// TwinCAT 3 PLC project PLC1
// ProgramVersion: 3.1.4026.16
// CompilerDefines: VISU_USEPROPERTYINFO
// libraries:
//   SH_Light, * (StroemHansen)
//   Tc2_EnOcean, * (Beckhoff Automation GmbH)
//   Tc2_Standard, * (Beckhoff Automation GmbH)
//   Tc2_System, * (Beckhoff Automation GmbH)
//   Tc2_Utilities, * (Beckhoff Automation GmbH)
//   Tc3_DALI, * (Beckhoff Automation GmbH)
//   Tc3_System_DK, * (Beckhoff - DK)
//   VisuDialogs, * (System)
// project tree:
//   DUTs/DALI/ E_DALIExtendedFadeTime.TcTLEO (not stored), ST_DALI102Parameters.TcDUT (not stored), ST_DALI103Parameters.TcDUT, ST_DALIMemoryBank.TcDUT (not stored), ST_DALI_GrpAssignment.TcDUT (not stored), ST_GroupSort.TcDUT (not stored)
//   DUTs/EnOcean/ ST_ReadSAB05.TcDUT (not stored), ST_WriteSAB05.TcDUT (not stored)
//   / FastTask.TcTTO (not stored), GlobalTextList.TcGTLO, PlcTask.TcTTO (not stored), Visualization Manager.TcVMO (not stored)
//   GVLs/ GVL_AHDataModbus.TcGVL (not stored), GVL_EnOcean.TcGVL, GVL_Skalering.TcGVL
//   POUs/01_System/01_System/GVLs/ GVL_EtherCAT.TcGVL (not stored)
//   POUs/01_System/01_System/ P_SystemDK.TcPOU (not stored)
//   POUs/AHModbusComm/ P_AHModbusComm.TcPOU
//   POUs/Alle_Rum/Gange/P_Gang_1_108/ P_Gang_1_108.TcPOU, Visualization_1_108.TcVIS (excluded from build)
//   POUs/Alle_Rum/Gange/P_Gang_1_111A/ P_Gang_1_111A.TcPOU, Visualization_1_111A.TcVIS (excluded from build)
//   POUs/Alle_Rum/Rum_Med_DALI_Pir/ P_Lys_Grp0.TcPOU (not stored) (excluded from build)
//   POUs/Alle_Rum/Rum_Med_DALI_Pir/Rum_1_111D/ P_Rum_1_111D.TcPOU, Visualization_1_111D.TcVIS (excluded from build)
//   POUs/Alle_Rum/Rum_Med_DALI_Pir/Rum_1_111E/ P_Rum_1_111E.TcPOU, Visualization_1.TcVIS (excluded from build)
//   POUs/Alle_Rum/Rum_Med_DALI_Pir/Rum_1_111C/ P_Rum_1_111C.TcPOU, Visualization_1_111C.TcVIS (excluded from build)
//   POUs/Alle_Rum/Rum_Med_DALI_Pir/Rum_1_115/ P_Rum_1_115.TcPOU, Visualization_1_115.TcVIS (excluded from build)
//   POUs/Alle_Rum/Rum_Med_DALI_Pir/Rum_1_118/ P_Rum_1_118.TcPOU, Visualization_1_118.TcVIS (excluded from build)
//   POUs/Alle_Rum/Rum_Med_DALI_Pir/Rum_1_106/ P_Rum_1_106.TcPOU, Visualization_1_106.TcVIS (excluded from build)
//   POUs/Alle_Rum/Trapper/ P_Trappe_T1.TcPOU
//   POUs/DALI/DALI_Setup/ DALI_Commissioning.TcPOU (not stored)
//   POUs/DALI/DALI_Setup/FBs/ FB_Part102Addressing.TcPOU (not stored), FB_Part102Commands.TcPOU (not stored), FB_Part102Groups.TcPOU (not stored), FB_Part102MemoryPages.TcPOU, FB_Part102Parameters.TcPOU, FB_Part102Scenes.TcPOU (not stored), FB_Part102SetFading.TcPOU, FB_Part103Addressing.TcPOU (not stored), FB_Part103MemoryPages.TcPOU (not stored), FB_Part103Identify.TcPOU (not stored), FB_Part103Parameters.TcPOU (not stored), FB_Part202Emergency.TcPOU (not stored), FB_Part205Incandescent.TcPOU (not stored), FB_Part207LED.TcPOU (not stored), FB_Part208Switching.TcPOU (not stored), FB_Part300GenericDevice.TcPOU (not stored), FB_Part301PushButton.TcPOU (not stored), FB_Part302AbsoluteInputDevice.TcPOU (not stored), FB_Part303OccupancySensor.TcPOU (not stored), FB_Part304LightSensor.TcPOU (not stored), GearType.TcPOU (not stored)
//   POUs/DALI/DALI_Setup/GVLs/ GVL_Internal.TcGVL (not stored)
//   POUs/DALI/DALI_Setup/VISUs/TextLists/ CommandOnTerminalEvent.TcTLO (not stored), DimmingCurve.TcTLO, EventPriority.TcTLO (not stored), EventScheme.TcTLO (not stored), ExtendedFadeTime.TcTLO (not stored), FadeRate.TcTLO (not stored), FadeTime.TcTLO (not stored), FastFadeTime.TcTLO (not stored), TextList_Dialogs.TcTLO (not stored)
//   POUs/DALI/DALI_Setup/VISUs/ Visu_DALICommissioning.TcVIS (not stored)
//   POUs/DALI/DALI_Setup/VISUs/Visu_DALICommissioning/ Visu_KL6821Configuration.TcVIS (not stored) (excluded from build), Visu_Part102Addressing.TcVIS (not stored), Visu_Part102Commands.TcVIS (not stored), Visu_Part102Groups.TcVIS (not stored), Visu_Part102MemoryBank.TcVIS, Visu_Part102Parameters.TcVIS, Visu_Part102Scenes.TcVIS (not stored), Visu_Part102SetFading.TcVIS (not stored), Visu_Part103Addressing.TcVIS (not stored), Visu_Part103MemoryBank.TcVIS, Visu_Part103Identify.TcVIS (not stored), Visu_Part103Parameters.TcVIS (not stored), Visu_Part202.TcVIS (not stored), Visu_Part202Commands.TcVIS, Visu_Part202Parameters.TcVIS (not stored), Visu_Part202Status.TcVIS (not stored), Visu_Part205.TcVIS (not stored), Visu_Part205Parameters.TcVIS (not stored), Visu_Part205Status.TcVIS, Visu_Part207.TcVIS (not stored), Visu_Part207Parameters.TcVIS (not stored), Visu_Part207Status.TcVIS, Visu_Part208Switching.TcVIS (not stored), Visu_Part300GenericDevice.TcVIS (not stored), Visu_Part301PushButton.TcVIS (not stored), Visu_Part302AbsoluteInputDevice.TcVIS, Visu_Part303OccupancySensor.TcVIS, Visu_Part304LightSensor.TcVIS, Visu_Welcome.TcVIS (not stored)
//   POUs/DALI/PRGs/Background/ P_DALI_Background.TcPOU (not stored)
//   POUs/DALI/PRGs/Diag/ P_DALI_DIAG.TcPOU (not stored)
//   POUs/DALI/PRGs/EnergyData/ P_DALI_Energy_Firmware_Test.TcPOU (not stored) (excluded from build), P_DALI_Energy_Line.TcPOU (not stored)
//   POUs/EnOcean/ P_EnOcean.TcPOU
//   POUs/ MAIN.TcPOU
//   POUs/Tester/ P_DALI2_Test.TcPOU (not stored) (excluded from build), P_Test_TypeA.TcPOU (not stored) (excluded from build), Visualization.TcVIS (excluded from build)
// real-time tasks:
//   TASK PlcTask: cycle T#40ms, priority 21, ADS port 350
//   TASK FastTask: cycle T#4ms, priority 20, ADS port 351
// I/O:
//   DEVICE Device 1 (Beckhoff CCAT)
//   DEVICE Device 3 (CX-BK)
//     Box 1 (CX-BK)
// variable links:
//   PLC1/PLC1 Instance <-> Device 3 (CX-BK)/Box 1 (CX-BK)
//     FastTask Inputs/P_DALI_Background.arrKL6821InData[1] @bit 16 <-> Term 5 (KL6821)/Channel 1/Data In 0
//     FastTask Inputs/P_DALI_Background.arrKL6821InData[1] @bit 24 <-> Term 5 (KL6821)/Channel 1/Data In 1
//     FastTask Inputs/P_DALI_Background.arrKL6821InData[1] @bit 32 <-> Term 5 (KL6821)/Channel 1/Data In 2
//     FastTask Inputs/P_DALI_Background.arrKL6821InData[1] @bit 40 <-> Term 5 (KL6821)/Channel 1/Data In 3
//     FastTask Inputs/P_DALI_Background.arrKL6821InData[2] @bit 16 <-> Term 6 (KL6821)/Channel 1/Data In 0
//     FastTask Inputs/P_DALI_Background.arrKL6821InData[2] @bit 24 <-> Term 6 (KL6821)/Channel 1/Data In 1
//     FastTask Inputs/P_DALI_Background.arrKL6821InData[2] @bit 32 <-> Term 6 (KL6821)/Channel 1/Data In 2
//     FastTask Inputs/P_DALI_Background.arrKL6821InData[2] @bit 40 <-> Term 6 (KL6821)/Channel 1/Data In 3
//     FastTask Inputs/P_DALI_Background.arrKL6821InData[1] <-> Term 5 (KL6821)/Channel 1/State
//     FastTask Inputs/P_DALI_Background.arrKL6821InData[2] <-> Term 6 (KL6821)/Channel 1/State
//     FastTask Inputs/P_EnOcean.stKL6581_in @bit 8 <-> Term 3 (KL6581)/Channel 1/Input CNODE
//     FastTask Inputs/P_EnOcean.stKL6581_in @bit {24..48 step 8} <-> Term 3 (KL6581)/Channel 1/Input DB{0..3}  (4 links)
//     FastTask Inputs/P_EnOcean.stKL6581_in @bit {56..80 step 8} <-> Term 3 (KL6581)/Channel 1/Input ID{0..3}  (4 links)
//     FastTask Inputs/P_EnOcean.stKL6581_in @bit 16 <-> Term 3 (KL6581)/Channel 1/Input ORG
//     FastTask Inputs/P_EnOcean.stKL6581_in @bit 88 <-> Term 3 (KL6581)/Channel 1/Input STATUS
//     FastTask Inputs/P_EnOcean.stKL6581_in <-> Term 3 (KL6581)/Channel 1/Status
//     FastTask Outputs/P_DALI_Background.arrKL6821OutData[1] <-> Term 5 (KL6821)/Channel 1/Ctrl
//     FastTask Outputs/P_DALI_Background.arrKL6821OutData[2] <-> Term 6 (KL6821)/Channel 1/Ctrl
//     FastTask Outputs/P_DALI_Background.arrKL6821OutData[1] @bit 16 <-> Term 5 (KL6821)/Channel 1/Data Out 0
//     FastTask Outputs/P_DALI_Background.arrKL6821OutData[1] @bit 24 <-> Term 5 (KL6821)/Channel 1/Data Out 1
//     FastTask Outputs/P_DALI_Background.arrKL6821OutData[1] @bit 32 <-> Term 5 (KL6821)/Channel 1/Data Out 2
//     FastTask Outputs/P_DALI_Background.arrKL6821OutData[1] @bit 40 <-> Term 5 (KL6821)/Channel 1/Data Out 3
//     FastTask Outputs/P_DALI_Background.arrKL6821OutData[2] @bit 16 <-> Term 6 (KL6821)/Channel 1/Data Out 0
//     FastTask Outputs/P_DALI_Background.arrKL6821OutData[2] @bit 24 <-> Term 6 (KL6821)/Channel 1/Data Out 1
//     FastTask Outputs/P_DALI_Background.arrKL6821OutData[2] @bit 32 <-> Term 6 (KL6821)/Channel 1/Data Out 2
//     FastTask Outputs/P_DALI_Background.arrKL6821OutData[2] @bit 40 <-> Term 6 (KL6821)/Channel 1/Data Out 3
//     FastTask Outputs/P_EnOcean.stKL6581_out <-> Term 3 (KL6581)/Channel 1/Control
//     FastTask Outputs/P_EnOcean.stKL6581_out @bit 8 <-> Term 3 (KL6581)/Channel 1/Output CNODE
//     FastTask Outputs/P_EnOcean.stKL6581_out @bit {24..48 step 8} <-> Term 3 (KL6581)/Channel 1/Output DB{0..3}  (4 links)
//     FastTask Outputs/P_EnOcean.stKL6581_out @bit {56..80 step 8} <-> Term 3 (KL6581)/Channel 1/Output ID{0..3}  (4 links)
//     FastTask Outputs/P_EnOcean.stKL6581_out @bit 16 <-> Term 3 (KL6581)/Channel 1/Output ORG
//     FastTask Outputs/P_EnOcean.stKL6581_out @bit 88 <-> Term 3 (KL6581)/Channel 1/Output STATUS
//     PlcTask Inputs/MAIN.nCX8200_State <-> Inputs/State
//     PlcTask Inputs/P_Trappe_T1.bDigitalPir <-> Term 4 (KL1408)/Channel 1/Input
//     PlcTask Outputs/P_Trappe_T1.bTrappelysNC <-> Term 2 (KL2012)/Channel 1/Output

// ---- DUTs/DALI/ST_DALI103Parameters.TcDUT
TYPE ST_DALI103Parameters :
STRUCT	
	//nShortAddress			:	BYTE;
	nOperatingMode			:	BYTE;
	sInstanceType0			:	STRING;	
	sInstanceType1			:	STRING;
	sInstanceType2			:	STRING;
	sInstanceType3			:	STRING;
	sInstanceType4			:	STRING;
END_STRUCT
END_TYPE

// ---- GVLs/GVL_EnOcean.TcGVL
{attribute 'qualified_only'}
VAR_GLOBAL
	strEnOceanSwitch_Gang_1_108: Tc2_EnOcean.STR_EnOceanSwitch;
	strEnOceanSwitch_Rum_1_106: Tc2_EnOcean.STR_EnOceanSwitch;
	strEnOceanSwitch_Rum_1_111E: Tc2_EnOcean.STR_EnOceanSwitch;
	strEnOceanSwitch_Rum_1_115_Gang: Tc2_EnOcean.STR_EnOceanSwitch;
	strEnOceanSwitch_Rum_1_115_Ydermur: Tc2_EnOcean.STR_EnOceanSwitch;
	strEnOceanSwitch_Rum_1_118: Tc2_EnOcean.STR_EnOceanSwitch;
	//strEnOceanSwitch_Rum_1_118: Tc2_EnOcean.STR_EnOceanSwitch;
END_VAR

// ---- GVLs/GVL_Skalering.TcGVL
//{attribute 'qualified_only'}
VAR_GLOBAL
fMeassure_Zone1 :REAL:= 604; 
fRead_Zone1     :REAL:= 340;

fMeassure_Zone2 :REAL:=611;
fRead_Zone2     :REAL:=374;

fMeassure_Zone3 :REAL:=986;
fRead_Zone3     :REAL:=524;

fMeassure_Zone4 :REAL:=770;
fRead_Zone4     :REAL:=506;

fMeassure_Zone5 :REAL:=734;
fRead_Zone5     :REAL:=395;

fMeassure_Zone6 :REAL:=890;
fRead_Zone6     :REAL:=476;

fMeassure_Zone7 :REAL:=710;
fRead_Zone7     :REAL:=654;

fMeassure_Zone8 :REAL:=604;
fRead_Zone8     :REAL:=292;

fMeassure_Zone9 :REAL:=572;
fRead_Zone9     :REAL:=348;

fMeassure_Zone10:REAL:= 790;
fRead_Zone10    :REAL:=434;

fMeassure_Zone11 :REAL:=691;
fRead_Zone11     :REAL:=426;

END_VAR

// ---- POUs/AHModbusComm/P_AHModbusComm.TcPOU
PROGRAM P_AHModbusComm
VAR
	arrfbReadAHPirData	: ARRAY[1..GVL_AHDataModbus.byNumberOfAH_Neighbors] OF SH_Light.FB_ReadAHPirData;
	arrReadAHPirData		: ARRAY[1..GVL_AHDataModbus.byNumberOfAH_Neighbors] OF BOOL;
	
	arrfbTriggerPulses			: ARRAY[1..GVL_AHDataModbus.byNumberOfAH_Neighbors] OF SH_Light.FB_ClockPulse;
	arrGeneratePulses			: ARRAY[1..GVL_AHDataModbus.byNumberOfAH_Neighbors] OF BOOL := [GVL_AHDataModbus.byNumberOfAH_Neighbors(TRUE)];
	tTimeInterval					: TIME := T#1S;
	tPulseTime					: TIME := T#1S;
	
	byLineId						: BYTE;
	byAHId						: BYTE;
		fbWritePirDelayTime		: R_TRIG;
	bRunOverrideOnce		: BOOL := FALSE;
	bEnableDelayTimeOverride : BOOL := FALSE;
	uiPirOffDelayTimeAllRooms : UINT := 30;
	
END_VAR

VAR CONSTANT
	arrnMBAddr					: ARRAY[1..GVL_AHDataModbus.byNumberOfAH_Neighbors] OF WORD := [GVL_AHDataModbus.byNumberOfAH_Neighbors(12588)]; //modbus-adresser (%MB600=>12588 default)
	arrstNeighborIPAddr		: ARRAY[1..GVL_AHDataModbus.byNumberOfAH_Neighbors] OF SH_Light.ST_NeighborIP := [
																						(sPLCName := 'AH1-1', sIP := '172.24.195.161', IsNeighbor := FALSE), 
																				     	(sPLCName := 'AH1-2', sIP := '172.24.195.162', IsNeighbor := FALSE), 
																						(sPLCName := 'AH1-3', sIP := '172.24.195.163', IsNeighbor := FALSE),
																						(sPLCName := 'AH2-1', sIP := '172.24.195.164', IsNeighbor := FALSE),
																					    (sPLCName := 'AH2-2', sIP := '172.24.195.165', IsNeighbor := FALSE),
																						(sPLCName := 'AH2-3', sIP := '172.24.195.166', IsNeighbor := FALSE),
																				        (sPLCName := 'AH2-4', sIP := '172.24.195.167', IsNeighbor := FALSE),
																						(sPLCName := 'AH2-5', sIP := '172.24.195.168', IsNeighbor := FALSE),
																						(sPLCName := 'AH3-2', sIP := '172.24.195.169', IsNeighbor := FALSE),
																						(sPLCName := 'AH3-3', sIP := '172.24.195.170', IsNeighbor := FALSE),
																			         	(sPLCName := 'AH3-4', sIP := '172.24.195.171', IsNeighbor := FALSE),
																						(sPLCName := 'AH3-5', sIP := '172.24.195.172', IsNeighbor := FALSE),
																						(sPLCName := 'AH4-1', sIP := '172.24.195.173', IsNeighbor := FALSE),
																						(sPLCName := 'AH4-2', sIP := '172.24.195.174', IsNeighbor := FALSE),
																						(sPLCName := 'AH4-3', sIP := '172.24.195.175', IsNeighbor := FALSE),
																			            (sPLCName := 'AH4-4', sIP := '172.24.195.176', IsNeighbor := FALSE),
																						(sPLCName := 'AH4-5', sIP := '172.24.195.177', IsNeighbor := FALSE),
																						(sPLCName := 'AH5-1', sIP := '172.24.195.178', IsNeighbor := FALSE),
																					    (sPLCName := 'AH5-2', sIP := '172.24.195.179', IsNeighbor := FALSE), 
																						(sPLCName := 'AH5-3', sIP := '172.24.195.180', IsNeighbor := FALSE),
																						(sPLCName := 'AH5-4', sIP := '172.24.195.181', IsNeighbor := FALSE),
																						(sPLCName := 'AH5-5', sIP := '172.24.195.182', IsNeighbor := FALSE),
																						(sPLCName := 'AH6-1', sIP := '172.24.195.183', IsNeighbor := FALSE),
																				        (sPLCName := 'AH6-2', sIP := '172.24.195.184', IsNeighbor := FALSE),//Local must be false
																				(sPLCName := 'AH6-3', sIP := '172.24.195.185', IsNeighbor := FALSE)];
																					//	(sPLCName := 'AH3-1', sIP := '172.24.195.186', IsNeighbor := TRUE) //when ready
END_VAR

A_AHNeighborRoomsPirIn();
A_AHNeighborRoomsPirOut();
A_DALILineShrtAddrErr();
A_DelayTimeAllRooms();

ACTION A_AHNeighborRoomsPirIn:
FOR byAHId := 1 TO GVL_AHDataModbus.byNumberOfAH_Neighbors DO
	IF arrstNeighborIPAddr[byAHId].IsNeighbor THEN
		//Generate Pulses
		arrfbTriggerPulses[byAHId](bGenerateClockPulses:= arrGeneratePulses[byAHId], tTimeInterval:= tTimeInterval, tPulseTime:= tPulseTime);
		arrReadAHPirData[byAHId]:= arrfbTriggerPulses[byAHId].bPulse;
		//Read data
		arrfbReadAHPirData[byAHId](	bReadAHPirData				:=	arrReadAHPirData[byAHId],
														sIPAddr							:=	arrstNeighborIPAddr[byAHId].sIP,
														nMBAddr							:=	arrnMBAddr[byAHId],
														nMBDataBuffer				:=	GVL_AHDataModbus.arrAH_NeighborRoomsPir_In[byAHId],
														arrAH_NeighborRoomsPir	=>GVL_AHDataModbus.arrAH_NeighborRoomsPir[byAHId]);
	END_IF
END_FOR
END_ACTION

ACTION A_AHNeighborRoomsPirOut:
//GVL_AHDataModbus.nAH_NeighborRoomsPir_Out.0 := P_Gang_4_413.bPirActive_MB;
//GVL_AHDataModbus.nAH_NeighborRoomsPir_Out.1 := P_Gang_7_401.bPirActive_MB;
//GVL_AHDataModbus.nAH_NeighborRoomsPir_Out.2 := P_Gang_5_441.bPirActive_MB;
//GVL_AHDataModbus.nAH_NeighborRoomsPir_Out.3 := P_Rum_4_424.bPirActive_MB;
//GVL_AHDataModbus.nAH_NeighborRoomsPir_Out.4 := P_Rum_4_426.bPirActive_MB;
//GVL_AHDataModbus.nAH_NeighborRoomsPir_Out.5 := 
//GVL_AHDataModbus.nAH_NeighborRoomsPir_Out.6 :=
//GVL_AHDataModbus.nAH_NeighborRoomsPir_Out.7 := 
//GVL_AHDataModbus.nAH_NeighborRoomsPir_Out.8 :=
//GVL_AHDataModbus.nAH_NeighborRoomsPir_Out.9 := 
//GVL_AHDataModbus.nAH_NeighborRoomsPir_Out.10 :=
//GVL_AHDataModbus.nAH_NeighborRoomsPir_Out.11 := 
//GVL_AHDataModbus.nAH_NeighborRoomsPir_Out.12 := 
//GVL_AHDataModbus.nAH_NeighborRoomsPir_Out.13 := 
//GVL_AHDataModbus.nAH_NeighborRoomsPir_Out.14 := 
//GVL_AHDataModbus.nAH_NeighborRoomsPir_Out.15 :=
END_ACTION

ACTION A_DALILineShrtAddrErr:
FOR  byLineId := 1 TO SH_Light.DALI_Param.MAX_DALIV2_LINES DO
	GVL_AHDataModbus.arrDALILineShrtAddrErr[byLineId] :=  TO_UINT(SH_Light.GVL_DALI_LatestError.arrLineShrtAddr[byLineId]);
END_FOR
END_ACTION

ACTION A_DelayTimeAllRooms:

fbWritePirDelayTime(CLK := GVL_AHDataModbus.uiPirOffDelayTimeAllRooms_MB<>uiPirOffDelayTimeAllRooms);

IF fbWritePirDelayTime.Q THEN
	bRunOverrideOnce := TRUE;
	bEnableDelayTimeOverride := TRUE;
	
//Indsæt kode
P_Gang_1_108.fbWritePirDelayTIme(bEnableOverride := bEnableDelayTimeOverride, nOverRideValue := GVL_AHDataModbus.uiPirOffDelayTimeAllRooms_MB, nValIn1 := GVL_AHDataModbus.uiPirOffDelayTimeAllRooms_MB, nValIn2 := uiPirOffDelayTimeAllRooms);
P_RUM_1_106.fbWritePirDelayTIme(bEnableOverride := bEnableDelayTimeOverride, nOverRideValue := GVL_AHDataModbus.uiPirOffDelayTimeAllRooms_MB, nValIn1 := GVL_AHDataModbus.uiPirOffDelayTimeAllRooms_MB, nValIn2 := uiPirOffDelayTimeAllRooms);
P_Rum_1_111E.fbWritePirDelayTIme(bEnableOverride := bEnableDelayTimeOverride, nOverRideValue := GVL_AHDataModbus.uiPirOffDelayTimeAllRooms_MB, nValIn1 := GVL_AHDataModbus.uiPirOffDelayTimeAllRooms_MB, nValIn2 := uiPirOffDelayTimeAllRooms);
P_Rum_1_115.fbWritePirDelayTIme(bEnableOverride := bEnableDelayTimeOverride, nOverRideValue := GVL_AHDataModbus.uiPirOffDelayTimeAllRooms_MB, nValIn1 := GVL_AHDataModbus.uiPirOffDelayTimeAllRooms_MB, nValIn2 := uiPirOffDelayTimeAllRooms);
P_Rum_1_118.fbWritePirDelayTIme(bEnableOverride := bEnableDelayTimeOverride, nOverRideValue := GVL_AHDataModbus.uiPirOffDelayTimeAllRooms_MB, nValIn1 := GVL_AHDataModbus.uiPirOffDelayTimeAllRooms_MB, nValIn2 := uiPirOffDelayTimeAllRooms);
P_Rum_1_111D.fbWritePirDelayTIme(bEnableOverride := bEnableDelayTimeOverride, nOverRideValue := GVL_AHDataModbus.uiPirOffDelayTimeAllRooms_MB, nValIn1 := GVL_AHDataModbus.uiPirOffDelayTimeAllRooms_MB, nValIn2 := uiPirOffDelayTimeAllRooms);
P_Gang_1_111A.fbWritePirDelayTIme(bEnableOverride := bEnableDelayTimeOverride, nOverRideValue := GVL_AHDataModbus.uiPirOffDelayTimeAllRooms_MB, nValIn1 := GVL_AHDataModbus.uiPirOffDelayTimeAllRooms_MB, nValIn2 := uiPirOffDelayTimeAllRooms);




ELSE
	IF bRunOverrideOnce THEN
		bEnableDelayTimeOverride := FALSE;
		
		//Indsæt kode
P_Gang_1_108.fbWritePirDelayTIme(bEnableOverride := bEnableDelayTimeOverride, nOverRideValue := GVL_AHDataModbus.uiPirOffDelayTimeAllRooms_MB, nValIn1 := GVL_AHDataModbus.uiPirOffDelayTimeAllRooms_MB, nValIn2 := uiPirOffDelayTimeAllRooms);
P_RUM_1_106.fbWritePirDelayTIme(bEnableOverride := bEnableDelayTimeOverride, nOverRideValue := GVL_AHDataModbus.uiPirOffDelayTimeAllRooms_MB, nValIn1 := GVL_AHDataModbus.uiPirOffDelayTimeAllRooms_MB, nValIn2 := uiPirOffDelayTimeAllRooms);
P_Rum_1_111E.fbWritePirDelayTIme(bEnableOverride := bEnableDelayTimeOverride, nOverRideValue := GVL_AHDataModbus.uiPirOffDelayTimeAllRooms_MB, nValIn1 := GVL_AHDataModbus.uiPirOffDelayTimeAllRooms_MB, nValIn2 := uiPirOffDelayTimeAllRooms);
P_Rum_1_115.fbWritePirDelayTIme(bEnableOverride := bEnableDelayTimeOverride, nOverRideValue := GVL_AHDataModbus.uiPirOffDelayTimeAllRooms_MB, nValIn1 := GVL_AHDataModbus.uiPirOffDelayTimeAllRooms_MB, nValIn2 := uiPirOffDelayTimeAllRooms);
P_Rum_1_118.fbWritePirDelayTIme(bEnableOverride := bEnableDelayTimeOverride, nOverRideValue := GVL_AHDataModbus.uiPirOffDelayTimeAllRooms_MB, nValIn1 := GVL_AHDataModbus.uiPirOffDelayTimeAllRooms_MB, nValIn2 := uiPirOffDelayTimeAllRooms);
P_Rum_1_111D.fbWritePirDelayTIme(bEnableOverride := bEnableDelayTimeOverride, nOverRideValue := GVL_AHDataModbus.uiPirOffDelayTimeAllRooms_MB, nValIn1 := GVL_AHDataModbus.uiPirOffDelayTimeAllRooms_MB, nValIn2 := uiPirOffDelayTimeAllRooms);
P_Gang_1_111A.fbWritePirDelayTIme(bEnableOverride := bEnableDelayTimeOverride, nOverRideValue := GVL_AHDataModbus.uiPirOffDelayTimeAllRooms_MB, nValIn1 := GVL_AHDataModbus.uiPirOffDelayTimeAllRooms_MB, nValIn2 := uiPirOffDelayTimeAllRooms);

		bRunOverrideOnce := FALSE;
		
		
	END_IF
END_IF
END_ACTION

END_PROGRAM

// ---- POUs/Alle_Rum/Gange/P_Gang_1_108/P_Gang_1_108.TcPOU
PROGRAM P_Gang_1_108
VAR
//Light

	fbLys		: FB_Light_Type_B;
	
	stDaliSetup	: SH_Light.ST_DALI_RoomSetup := (		byShrtAdr_Prim := 25, 
														byGrpAdr_Prim := 4, 
														eMod_Prim := E_DALIAddressType.Group, 
														//byShrtAdr_Sec := 1, 
														//byGrpAdr_Sec := 1, 
														//eMod_Sec := E_DALIAddressType.Short, 
														//byShrtAdr_Supl := 1, 
														DALI_LINE_NUM_PRIM := 1, 
														DALI_LINE_NUM_SEC := 0, 
														DALI_LINE_NUM_SUPL := 0);
	stLiveData				: SH_Light.ST_LiveData;
	bRunTuning					: BOOL;
	
	bTopButtonZone1				: BOOL;
	bTopButtonZone1_Visu		: BOOL;
	bBottomButtonZone1			: BOOL;
	bBottomButtonZone1_Visu	    : BOOL;
	bButtonZone2				: BOOL;
	bNeighborRoomsPir		    : BOOL;
	fLuxOn				     	: REAL;
	fLuxDim						: REAL;
	tPIRDim						: TIME;
	tPIROff						: TIME;
	fOffsetSec					: REAL := 20;
	bOccupiedRoom			    : BOOL;



// Sensor Settings	
	fbSensor					: SH_Light.FB_NIKO_P46xx_2Pcs;
	//fbSensor					: SH_Light.FB_NIKO_P46xx_2Pcs;
	//bySensorAddr				: BYTE := 3;
	arrSensorAddr				: ARRAY[1..2] OF BYTE := [7,8];
	bInitialize					: BOOL := TRUE;
	stDaliSensorSetup			: ST_DALI_NIKOP46SetupData := (
																nSensitivityPIRSegmentA := arrSensitivityOccupancy[1],
																nSensitivityPIRSegmentB := arrSensitivityOccupancy[2],
																nSensitivityPIRSegmentC := arrSensitivityOccupancy[3]);

	//bInitErr				: BOOL;
	//bInitDone				: BOOL;
	arrInitErr					: ARRAY [1..2] OF BOOL;
	arrInitDone					: ARRAY [1..2] OF BOOL;
	arrSensorScales				: ARRAY [1..10] OF SH_Light.ST_DALI_SensorScaleMode := [	(fMeassureMaxSensor := fMeassure_Zone4, fReadMaxSensor := fRead_Zone4),
																							(fMeassureMaxSensor := fMeassure_Zone4, fReadMaxSensor := fRead_Zone4),
																						8(())];
	bCancelHoldTimerOccupancy	: BOOL;
(*	eEventPriorityOccupancy		: E_DALIEventPriority := E_DALIEVENTPRIORITY.Middle;
	nHoldTimerOccupancy			: WORD := 5; // Value in s. 	
	nReportTimerOccupancy		: BYTE := 120; // Value in s, Preset manufacturer value
	nDeadtimeTimerOccupancy		: WORD := 100; // Value in ms, Predefined Value of DALI Standard
	bCancelHoldTimerOccupancy	: BOOL;
	nSensitivityOccupancy		: BYTE:= 3; //setting Sensivity (0..4) 0 (Off), 1 (Min), 2(Low), 3(High) and 4 (Max)

	bEnableLuxEvent				: BOOL;
	eEventPriorityBrightness	: E_DALIEventPriority := E_DALIEVENTPRIORITY.Middle;
	nDeadtimeTimerBrightness	: WORD := 1500; // Value in ms, Predefined Value of DALI Standard
	nHysteresisBrightness		: BYTE := 2; // Value in %
	nHysteresisMinBrightness	: BYTE := 10; // Absolute Value, depending on the manufacturer specific resolution
	nReportTimerBrightness		: BYTE := 120; // Value in s, Preset manufacturer value
*)

	//ModbusComm setup
	
	fbWriteSPLuxLevel			: SH_Light.FB_TwoVal_SelectOne_RTrigChange;
	fbWritePirDelayTIme		: SH_Light.FB_TwoVal_SelectOne_RTrigChange;
	stRoomDataPLC				: SH_Light.ST_RoomDataPLC	:=	(
																	uiPirOffDelayTime	:= 30,
																	uiSpLuxLevel		:= 500,
																	uiPirDimDelayTime	:= 15,
																	uiSpDimLuxLevel		:= 200);
																	
	fbBallastOnHours				: SH_Light.FB_CountOnHours;
	bEnableHourCount			: BOOL := TRUE;
	
	//Non-persistent modbus data
	bPirActive_MB					AT %MX16.0	: BOOL;				//bPirLys i gammel kode
	uiActLuxLevel_MB			    AT %MB20	: UINT;				//intHMIAktueltLux i gammel kode
	uiActLightLevelPct_MB	        AT %MB24	: UINT;				//intDALI_Gruppe1_Lysniveau i gammel kode
	
	//For Conversion
	uiPirOffMinutes						: UINT;
	udTimeScaling						: UDINT := 60000;
	uiLuxOn								: UINT;
	
	//max values checks
	uiMaxLuxLevel						: UINT := 1023;
	uiMaxPirOffMinutes				    : UINT := 180;



END_VAR

VAR CONSTANT
	Sesnor_DALI_LINE_NUM: BYTE := 2;
	DALI_LINE_NUM_LIGHT: BYTE:= 1;
	DALI_LINE_NUM_PENDANTS	            : BYTE := 0; //0=ingen pendler	
	arrSensitivityOccupancy				: ARRAY[1..3] OF BYTE := [4,4,4]; //sensitivitet for sensor

END_VAR
VAR PERSISTENT
	stPirSensorData: SH_Light.ST_DALI_Sensor;
	stTuneData: SH_Light.ST_TuneData_EX;
	
	
	uiPirOffDelayTime_MB	AT %MB18	: UINT;				//ntHMI_Pir_SetValue i gammel kode
	uiSPLuxLevel_MB			AT %MB22	: UINT;				//intHMI_Lux_SetValue i gammel kode
	uiBallastOnHours_MB		AT %MB26	: UINT;				//dintHMILysbraendtimer1 i gammel kode
	byOnHoursOverflowCount				: BYTE;   

END_VAR

A_Buttons();
A_LightCtrl();
A_Sensor();
A_Modbuscomm();

ACTION A_Buttons:
bTopButtonZone1		:= GVL_EnOcean.strEnOceanSwitch_Gang_1_108.bT1_ON OR bTopButtonZone1_Visu;
bBottomButtonZone1	:= GVL_EnOcean.strEnOceanSwitch_Gang_1_108.bT1_OFF OR bBottomButtonZone1_Visu;
;
END_ACTION

ACTION A_LightCtrl:
bNeighborRoomsPir	:= P_Rum_1_106.stPirSensorData.bPrc OR P_Rum_1_115.stPirSensorData.bPrc OR P_Rum_1_118.stPirSensorData.bPrc OR P_gang_1_111A.stPirSensorData.bPrc;
fbLys( 
	nZoneID:= 1, 
	bButtonZone1:= bTopButtonZone1,
	bBottomButtonZone1 := bBottomButtonZone1, 
	//bButtonZone2:= bButtonZone2,
	bNeighborRoomsPir	:=	bNeighborRoomsPir,
	fLuxOn:= fLuxOn, 
	fLuxDim:= fLuxDim, 
	tPIRDim:= tPIRDim, 
	tPIROff:= tPIROff, 
	fOffsetSec:= fOffsetSec, 
	bReInit:= , 
	stDaliSetup:= stDaliSetup, 
	ipCommunication_Prim:= P_DALI_Background.arrfbKL6821Communication[DALI_LINE_NUM_LIGHT], 
	//ipCommunication_Sec:= P_DALI_Background.arrfbKL6821Communication[DALI_LINE_NUM_LIGHT], 
	//ipCommunication_Supl:= P_DALI_Background.arrfbKL6821Communication[DALI_LINE_NUM_LIGHT], 
	fMinOutputPowerLevelRoom:= 15, 
	fMaxOutputPowerLevelRoom:= 100, 
	nCycleTimeInMS:= SH_Light.DALI_Param.nPlcTaskCycleTimeInMS*nDimCmdCycleTimeFactor , 
	bRunTuning:= bRunTuning, 
	bOccupiedRoom=> bOccupiedRoom, 
	bError_Prim=> , 
	nError_Prim=> , 
	stTuneData:=stTuneData , 
	stPirSensorData:= stPirSensorData, 
	stLiveData:= stLiveData);
END_ACTION

ACTION A_ModbusComm:
//Manage data for modbus communication

//Manage data for read-only in PLC
stRoomDataPLC.bPirActive			:= stPirSensorData.bPrc;
stRoomDataPLC.uiActLuxLevel			:= TO_UINT(TRUNC(stPirSensorData.fBrightness));
stRoomDataPLC.uiActLightLevelPct	:= TO_UINT(TRUNC(fbLys.fbBallast.fActlLgtLvl_Prim));
		//stRoomDataPLC.uiActLightLevelPct	:= TO_UINT(TRUNC(fbLys.fbBallast.fActlLgtLvl_Prim)); //if only one group light control
stRoomDataPLC.uiBallastOnHours		:= uiBallastOnHours_MB; //The calculation for BallastOnHours is stored directly to the MB register below


//Assign data for read-only to MB registers
bPirActive_MB			:= stRoomDataPLC.bPirActive;
uiActLuxLevel_MB		:= stRoomDataPLC.uiActLuxLevel;
uiActLightLevelPct_MB	:= stRoomDataPLC.uiActLightLevelPct;

	//calculate BallastOnHours
	fbBallastOnHours(
		bEnableHourCount	:= bEnableHourCount,
		bPauseCount			:= fbLys.fbLightCtrl.bOffZone1,
		uiOnHours			:= uiBallastOnHours_MB,			//OnHours is updated here
		byOverflowCount		:= byOnHoursOverflowCount);


//Manage data for read/write for both PLC and MB registers
fbWriteSPLuxLevel(	nMaxValOut	:= uiMaxLuxLevel,
					nValIn1		:= uiSPLuxLevel_MB,		//nValIn1 takes priotity in case of download or restart
					nValIn2		:= stRoomDataPLC.uiSpLuxLevel,
					nValOut		=> uiLuxOn
				);


fbWritePirDelayTIme(	nMaxValOut	:= uiMaxPirOffMinutes,
						nValIn1		:= uiPirOffDelayTime_MB,		//nValIn1 takes priotity in case of download or restart
						nValIn2		:= stRoomDataPLC.uiPirOffDelayTime,
						nValOut		=> uiPirOffMinutes
					);
					

//Convert read/write modbus data to appropriate datatypes in PLC
fLuxOn	:= TO_REAL(uiLuxOn);			
tPIROff	:= TO_TIME(uiPirOffMinutes*udTimeScaling); //Time conversion defaults to ms

fLuxDim	:= TO_REAL(stRoomDataPLC.uiSpDimLuxLevel);			
tPIRDim	:= TO_TIME(stRoomDataPLC.uiPirDimDelayTime*udTimeScaling); //Time conversion defaults to ms
END_ACTION

ACTION A_Sensor:

fbSensor.ipCommunication := P_DALI_Background.arrfbKL6821Communication[Sesnor_DALI_LINE_NUM];

fbSensor(
	arrShrtAdr:= arrSensorAddr,
	bInitialize:= bInitialize, 
	DALI_LINE_NUM:= Sesnor_DALI_LINE_NUM, 
 	//bCancelHoldTimerOccupancy:= bCancelHoldTimerOccupancy, 
	stSensorSetup := stDaliSensorSetup,
	arrInitErr=> arrInitErr, 
	arrInitDone=> arrInitDone,
	stPirSensorData:= stPirSensorData, 
	arrSensorScales:= arrSensorScales);
END_ACTION

END_PROGRAM

// ---- POUs/Alle_Rum/Rum_Med_DALI_Pir/Rum_1_106/P_Rum_1_106.TcPOU
PROGRAM P_Rum_1_106
VAR
//Light

	fbLys		: FB_Light_Type_A;
	
	stDaliSetup	: SH_Light.ST_DALI_RoomSetup := (		byShrtAdr_Prim := 32, 
														byGrpAdr_Prim := 5, 
														eMod_Prim := E_DALIAddressType.Group, 
														//byShrtAdr_Sec := 1, 
														//byGrpAdr_Sec := 1, 
														//eMod_Sec := E_DALIAddressType.Short, 
														//byShrtAdr_Supl := 1, 
														DALI_LINE_NUM_PRIM := 1, 
														DALI_LINE_NUM_SEC := 0, 
														DALI_LINE_NUM_SUPL := 0);
	stLiveData				: SH_Light.ST_LiveData;
	bRunTuning					: BOOL;
	
	bTopButtonZone1				: BOOL;
	bTopButtonZone1_Visu		: BOOL;
	bBottomButtonZone1			: BOOL;
	bBottomButtonZone1_Visu	    : BOOL;
	bButtonZone2				: BOOL;
	bNeighborRoomsPir		    : BOOL;
	fLuxOn				     	: REAL;
	fLuxDim						: REAL;
	tPIRDim						: TIME;
	tPIROff						: TIME;
	fOffsetSec					: REAL := 20;
	bOccupiedRoom			    : BOOL;

// Sensor Settings	
	fbSensor					: SH_Light.FB_NIKO_P46xx_2Pcs;
	//fbSensor					: SH_Light.FB_NIKO_P46xx_2Pcs;
	//bySensorAddr				: BYTE := 3;
	arrSensorAddr				: ARRAY[1..2] OF BYTE := [9,10];
	bInitialize					: BOOL := TRUE;
	stDaliSensorSetup			: ST_DALI_NIKOP46SetupData := (
																nSensitivityPIRSegmentA := arrSensitivityOccupancy[1],
																nSensitivityPIRSegmentB := arrSensitivityOccupancy[2],
																nSensitivityPIRSegmentC := arrSensitivityOccupancy[3]);

	//bInitErr				: BOOL;
	//bInitDone				: BOOL;
	arrInitErr					: ARRAY [1..2] OF BOOL;
	arrInitDone					: ARRAY [1..2] OF BOOL;
	arrSensorScales				: ARRAY [1..10] OF SH_Light.ST_DALI_SensorScaleMode := [	(fMeassureMaxSensor := fMeassure_Zone1, fReadMaxSensor := fRead_Zone1),
																							(fMeassureMaxSensor := fMeassure_Zone1, fReadMaxSensor := fRead_Zone1),
																						8(())];
	bCancelHoldTimerOccupancy	: BOOL;
(*	eEventPriorityOccupancy		: E_DALIEventPriority := E_DALIEVENTPRIORITY.Middle;
	nHoldTimerOccupancy			: WORD := 5; // Value in s. 	
	nReportTimerOccupancy		: BYTE := 120; // Value in s, Preset manufacturer value
	nDeadtimeTimerOccupancy		: WORD := 100; // Value in ms, Predefined Value of DALI Standard
	bCancelHoldTimerOccupancy	: BOOL;
	nSensitivityOccupancy		: BYTE:= 3; //setting Sensivity (0..4) 0 (Off), 1 (Min), 2(Low), 3(High) and 4 (Max)

	bEnableLuxEvent				: BOOL;
	eEventPriorityBrightness	: E_DALIEventPriority := E_DALIEVENTPRIORITY.Middle;
	nDeadtimeTimerBrightness	: WORD := 1500; // Value in ms, Predefined Value of DALI Standard
	nHysteresisBrightness		: BYTE := 2; // Value in %
	nHysteresisMinBrightness	: BYTE := 10; // Absolute Value, depending on the manufacturer specific resolution
	nReportTimerBrightness		: BYTE := 120; // Value in s, Preset manufacturer value
*)

	//ModbusComm setup
	
	fbWriteSPLuxLevel			: SH_Light.FB_TwoVal_SelectOne_RTrigChange;
	fbWritePirDelayTIme		: SH_Light.FB_TwoVal_SelectOne_RTrigChange;
	stRoomDataPLC				: SH_Light.ST_RoomDataPLC	:=	(
																	uiPirOffDelayTime	:= 30,
																	uiSpLuxLevel		:= 500,
																	uiPirDimDelayTime	:= 15,
																	uiSpDimLuxLevel		:= 200);
																	
	fbBallastOnHours				: SH_Light.FB_CountOnHours;
	bEnableHourCount			: BOOL := TRUE;
	
	//Non-persistent modbus data
	bPirActive_MB					AT %MX0.0	: BOOL;				//bPirLys i gammel kode
	uiActLuxLevel_MB			    AT %MB4	: UINT;				//intHMIAktueltLux i gammel kode
	uiActLightLevelPct_MB	        AT %MB8	: UINT;				//intDALI_Gruppe1_Lysniveau i gammel kode
	
	//For Conversion
	uiPirOffMinutes						: UINT;
	udTimeScaling						: UDINT := 60000;
	uiLuxOn								: UINT;
	
	//max values checks
	uiMaxLuxLevel						: UINT := 1023;
	uiMaxPirOffMinutes				    : UINT := 180;

	
END_VAR

VAR CONSTANT
	Sesnor_DALI_LINE_NUM: BYTE := 2;
	DALI_LINE_NUM_LIGHT: BYTE := 1;
	DALI_LINE_NUM_PENDANTS	            : BYTE := 0; //0=ingen pendler	
	arrSensitivityOccupancy				: ARRAY[1..3] OF BYTE := [4,4,4]; //sensitivitet for sensor

END_VAR
VAR PERSISTENT
	stPirSensorData: SH_Light.ST_DALI_Sensor;
	stTuneData: SH_Light.ST_TuneData_EX;
	
	uiPirOffDelayTime_MB	AT %MB2	: UINT;				//ntHMI_Pir_SetValue i gammel kode
	uiSPLuxLevel_MB			AT %MB6	: UINT;				//intHMI_Lux_SetValue i gammel kode
	uiBallastOnHours_MB		AT %MB10	: UINT;				//dintHMILysbraendtimer1 i gammel kode
	byOnHoursOverflowCount				: BYTE;   

END_VAR

A_Buttons();
A_LightCtrl();
A_Sensor();
A_modBuscomm();

ACTION A_Buttons:
bTopButtonZone1		:= GVL_EnOcean.strEnOceanSwitch_Rum_1_106.bT2_ON OR bTopButtonZone1_Visu;
bBottomButtonZone1	:= GVL_EnOcean.strEnOceanSwitch_Rum_1_106.bT2_OFF OR bBottomButtonZone1_Visu;
END_ACTION

ACTION A_LightCtrl:

fbLys(
	nZoneID:= 1, 
	bButtonZone1:= bTopButtonZone1,
	bBottomButtonZone1 := bBottomButtonZone1, 
	//bButtonZone2:= bButtonZone2, 
	fLuxOn:= fLuxOn, 
	fLuxDim:= fLuxDim, 
	tPIRDim:= tPIRDim, 
	tPIROff:= tPIROff, 
	fOffsetSec:= fOffsetSec, 
	bReInit:= , 
	stDaliSetup:= stDaliSetup, 
	ipCommunication_Prim:= P_DALI_Background.arrfbKL6821Communication[DALI_LINE_NUM_LIGHT], 
	//ipCommunication_Sec:= P_DALI_Background.arrfbKL6821Communication[DALI_LINE_NUM_LIGHT], 
	//ipCommunication_Supl:= P_DALI_Background.arrfbKL6821Communication[DALI_LINE_NUM_LIGHT], 
	fMinOutputPowerLevelRoom:= 15, 
	fMaxOutputPowerLevelRoom:= 100, 
	nCycleTimeInMS:= SH_Light.DALI_Param.nPlcTaskCycleTimeInMS*nDimCmdCycleTimeFactor , 
	bRunTuning:= bRunTuning, 
	bOccupiedRoom=> bOccupiedRoom, 
	bError_Prim=> , 
	nError_Prim=> , 
	stTuneData:=stTuneData , 
	stPirSensorData:= stPirSensorData, 
	stLiveData:= stLiveData);
END_ACTION

ACTION A_ModbusComm:
//Manage data for modbus communication

//Manage data for read-only in PLC
stRoomDataPLC.bPirActive			:= stPirSensorData.bPrc;
stRoomDataPLC.uiActLuxLevel			:= TO_UINT(TRUNC(stPirSensorData.fBrightness));
stRoomDataPLC.uiActLightLevelPct	:= TO_UINT(TRUNC(fbLys.fbBallast.fActlLgtLvl_Prim));
		//stRoomDataPLC.uiActLightLevelPct	:= TO_UINT(TRUNC(fbLys.fbBallast.fActlLgtLvl_Prim)); //if only one group light control
stRoomDataPLC.uiBallastOnHours		:= uiBallastOnHours_MB; //The calculation for BallastOnHours is stored directly to the MB register below


//Assign data for read-only to MB registers
bPirActive_MB			:= stRoomDataPLC.bPirActive;
uiActLuxLevel_MB		:= stRoomDataPLC.uiActLuxLevel;
uiActLightLevelPct_MB	:= stRoomDataPLC.uiActLightLevelPct;

	//calculate BallastOnHours
	fbBallastOnHours(
		bEnableHourCount	:= bEnableHourCount,
		bPauseCount			:= fbLys.fbLightCtrl.bOffZone1,
		uiOnHours			:= uiBallastOnHours_MB,			//OnHours is updated here
		byOverflowCount		:= byOnHoursOverflowCount);


//Manage data for read/write for both PLC and MB registers
fbWriteSPLuxLevel(	nMaxValOut	:= uiMaxLuxLevel,
					nValIn1		:= uiSPLuxLevel_MB,		//nValIn1 takes priotity in case of download or restart
					nValIn2		:= stRoomDataPLC.uiSpLuxLevel,
					nValOut		=> uiLuxOn
				);


fbWritePirDelayTIme(	nMaxValOut	:= uiMaxPirOffMinutes,
						nValIn1		:= uiPirOffDelayTime_MB,		//nValIn1 takes priotity in case of download or restart
						nValIn2		:= stRoomDataPLC.uiPirOffDelayTime,
						nValOut		=> uiPirOffMinutes
					);
					

//Convert read/write modbus data to appropriate datatypes in PLC
fLuxOn	:= TO_REAL(uiLuxOn);			
tPIROff	:= TO_TIME(uiPirOffMinutes*udTimeScaling); //Time conversion defaults to ms

fLuxDim	:= TO_REAL(stRoomDataPLC.uiSpDimLuxLevel);			
tPIRDim	:= TO_TIME(stRoomDataPLC.uiPirDimDelayTime*udTimeScaling); //Time conversion defaults to ms
END_ACTION

ACTION A_Sensor:

fbSensor.ipCommunication := P_DALI_Background.arrfbKL6821Communication[Sesnor_DALI_LINE_NUM];

fbSensor(
	arrShrtAdr:= arrSensorAddr,
	bInitialize:= bInitialize, 
	DALI_LINE_NUM:= Sesnor_DALI_LINE_NUM, 
 	//bCancelHoldTimerOccupancy:= bCancelHoldTimerOccupancy, 
	stSensorSetup := stDaliSensorSetup,
	arrInitErr=> arrInitErr, 
	arrInitDone=> arrInitDone,
	stPirSensorData:= stPirSensorData, 
	arrSensorScales:= arrSensorScales);
END_ACTION

END_PROGRAM

// ---- POUs/Alle_Rum/Rum_Med_DALI_Pir/Rum_1_115/P_Rum_1_115.TcPOU
PROGRAM P_Rum_1_115
VAR
//Light

	fbLys		: FB_Light_Type_A;
	
	stDaliSetup	: SH_Light.ST_DALI_RoomSetup := (		byShrtAdr_Prim := 3, 
														byGrpAdr_Prim := 2, 
														eMod_Prim := E_DALIAddressType.Group, 
														//byShrtAdr_Sec := 1, 
														//byGrpAdr_Sec := 1, 
														//eMod_Sec := E_DALIAddressType.Short, 
														//byShrtAdr_Supl := 1, 
														DALI_LINE_NUM_PRIM := 1, 
														DALI_LINE_NUM_SEC := 0, 
														DALI_LINE_NUM_SUPL := 0);
	stLiveData				: SH_Light.ST_LiveData;
bRunTuning					: BOOL;
	
	bTopButtonZone1				: BOOL;
	bTopButtonZone1_Visu		: BOOL;
	bBottomButtonZone1			: BOOL;
	bBottomButtonZone1_Visu	    : BOOL;
	bButtonZone2				: BOOL;
	bNeighborRoomsPir		    : BOOL;
	fLuxOn				     	: REAL;
	fLuxDim						: REAL;
	tPIRDim						: TIME;
	tPIROff						: TIME;
	fOffsetSec					: REAL := 20;
	bOccupiedRoom			    : BOOL;



// Sensor Settings	
	fbSensor					: SH_Light.FB_NIKO_P46xx_3Pcs;
	//fbSensor					: SH_Light.FB_NIKO_P46xx_2Pcs;
	//bySensorAddr				: BYTE := 3;
	arrSensorAddr				: ARRAY[1..3] OF BYTE := [2,3,4];
	bInitialize					: BOOL := TRUE;
	stDaliSensorSetup			: ST_DALI_NIKOP46SetupData;
	//bInitErr				: BOOL;
	//bInitDone				: BOOL;
	arrInitErr					: ARRAY [1..3] OF BOOL;
	arrInitDone					: ARRAY [1..3] OF BOOL;
	arrSensorScales				: ARRAY [1..10] OF SH_Light.ST_DALI_SensorScaleMode := [	(fMeassureMaxSensor := fMeassure_Zone3, fReadMaxSensor := fRead_Zone3),
																							(fMeassureMaxSensor := fMeassure_Zone3, fReadMaxSensor := fRead_Zone3),
																							(fMeassureMaxSensor := fMeassure_Zone3, fReadMaxSensor := fRead_Zone3),
																						7(())];
	bCancelHoldTimerOccupancy	: BOOL;
(*	eEventPriorityOccupancy		: E_DALIEventPriority := E_DALIEVENTPRIORITY.Middle;
	nHoldTimerOccupancy			: WORD := 5; // Value in s. 	
	nReportTimerOccupancy		: BYTE := 120; // Value in s, Preset manufacturer value
	nDeadtimeTimerOccupancy		: WORD := 100; // Value in ms, Predefined Value of DALI Standard
	bCancelHoldTimerOccupancy	: BOOL;
	nSensitivityOccupancy		: BYTE:= 3; //setting Sensivity (0..4) 0 (Off), 1 (Min), 2(Low), 3(High) and 4 (Max)

	bEnableLuxEvent				: BOOL;
	eEventPriorityBrightness	: E_DALIEventPriority := E_DALIEVENTPRIORITY.Middle;
	nDeadtimeTimerBrightness	: WORD := 1500; // Value in ms, Predefined Value of DALI Standard
	nHysteresisBrightness		: BYTE := 2; // Value in %
	nHysteresisMinBrightness	: BYTE := 10; // Absolute Value, depending on the manufacturer specific resolution
	nReportTimerBrightness		: BYTE := 120; // Value in s, Preset manufacturer value
*)

	//ModbusComm setup
	
	fbWriteSPLuxLevel			: SH_Light.FB_TwoVal_SelectOne_RTrigChange;
	fbWritePirDelayTIme		: SH_Light.FB_TwoVal_SelectOne_RTrigChange;
	stRoomDataPLC				: SH_Light.ST_RoomDataPLC	:=	(
																	uiPirOffDelayTime	:= 30,
																	uiSpLuxLevel		:= 500,
																	uiPirDimDelayTime	:= 15,
																	uiSpDimLuxLevel		:= 200);
																	
	fbBallastOnHours				: SH_Light.FB_CountOnHours;
	bEnableHourCount			: BOOL := TRUE;
	
	//Non-persistent modbus data
	bPirActive_MB					AT %MX48.0	: BOOL;				//bPirLys i gammel kode
	uiActLuxLevel_MB			    AT %MB52	: UINT;				//intHMIAktueltLux i gammel kode
	uiActLightLevelPct_MB	        AT %MB56	: UINT;				//intDALI_Gruppe1_Lysniveau i gammel kode
	
	//For Conversion
	uiPirOffMinutes						: UINT;
	udTimeScaling						: UDINT := 60000;
	uiLuxOn								: UINT;
	
	//max values checks
	uiMaxLuxLevel						: UINT := 1023;
	uiMaxPirOffMinutes				    : UINT := 180;

END_VAR

VAR CONSTANT
	Sesnor_DALI_LINE_NUM: BYTE := 2;
	DALI_LINE_NUM_LIGHT: BYTE := 1;
	DALI_LINE_NUM_PENDANTS	            : BYTE := 0; //0=ingen pendler	
	arrSensitivityOccupancy				: ARRAY[1..3] OF BYTE := [4,4,4]; //sensitivitet for sensor

END_VAR
VAR PERSISTENT
	stPirSensorData: SH_Light.ST_DALI_Sensor;
	stTuneData: SH_Light.ST_TuneData_EX;
	
	uiPirOffDelayTime_MB	AT %MB50	: UINT;				//ntHMI_Pir_SetValue i gammel kode
	uiSPLuxLevel_MB			AT %MB54	: UINT;				//intHMI_Lux_SetValue i gammel kode
	uiBallastOnHours_MB		AT %MB58	: UINT;				//dintHMILysbraendtimer1 i gammel kode
	byOnHoursOverflowCount				: BYTE;   

END_VAR

A_Buttons();
A_LightCtrl();
A_Sensor();
A_Modbuscomm();

ACTION A_Buttons:
bTopButtonZone1		:= GVL_EnOcean.strEnOceanSwitch_Rum_1_115_Gang.bT1_ON OR GVL_EnOcean.strEnOceanSwitch_Rum_1_115_Ydermur.bT1_ON OR bTopButtonZone1_Visu;
bBottomButtonZone1	:= GVL_EnOcean.strEnOceanSwitch_Rum_1_115_Gang.bT1_OFF OR GVL_EnOcean.strEnOceanSwitch_Rum_1_115_Ydermur.bT1_OFF OR bBottomButtonZone1_Visu;
END_ACTION

ACTION A_LightCtrl:

fbLys(
	nZoneID:= 1, 
	bButtonZone1:= bTopButtonZone1,
	bBottomButtonZone1 := bBottomButtonZone1, 
	bButtonZone2:= bButtonZone2, 
	fLuxOn:= fLuxOn, 
	fLuxDim:= fLuxDim, 
	tPIRDim:= tPIRDim, 
	tPIROff:= tPIROff, 
	fOffsetSec:= fOffsetSec, 
	bReInit:= , 
	stDaliSetup:= stDaliSetup, 
	ipCommunication_Prim:= P_DALI_Background.arrfbKL6821Communication[DALI_LINE_NUM_LIGHT], 
	//ipCommunication_Sec:= P_DALI_Background.arrfbKL6821Communication[DALI_LINE_NUM_LIGHT], 
	//ipCommunication_Supl:= P_DALI_Background.arrfbKL6821Communication[DALI_LINE_NUM_LIGHT], 
	fMinOutputPowerLevelRoom:= 15, 
	fMaxOutputPowerLevelRoom:= 100, 
	nCycleTimeInMS:= SH_Light.DALI_Param.nPlcTaskCycleTimeInMS*nDimCmdCycleTimeFactor , 
	bRunTuning:= bRunTuning, 
	bOccupiedRoom=> bOccupiedRoom, 
	bError_Prim=> , 
	nError_Prim=> , 
	stTuneData:=stTuneData , 
	stPirSensorData:= stPirSensorData, 
	stLiveData:= stLiveData);
END_ACTION

ACTION A_ModbusComm:
//Manage data for modbus communication

//Manage data for read-only in PLC
stRoomDataPLC.bPirActive			:= stPirSensorData.bPrc;
stRoomDataPLC.uiActLuxLevel			:= TO_UINT(TRUNC(stPirSensorData.fBrightness));
stRoomDataPLC.uiActLightLevelPct	:= TO_UINT(TRUNC(fbLys.fbBallast.fActlLgtLvl_Prim));
		//stRoomDataPLC.uiActLightLevelPct	:= TO_UINT(TRUNC(fbLys.fbBallast.fActlLgtLvl_Prim)); //if only one group light control
stRoomDataPLC.uiBallastOnHours		:= uiBallastOnHours_MB; //The calculation for BallastOnHours is stored directly to the MB register below


//Assign data for read-only to MB registers
bPirActive_MB			:= stRoomDataPLC.bPirActive;
uiActLuxLevel_MB		:= stRoomDataPLC.uiActLuxLevel;
uiActLightLevelPct_MB	:= stRoomDataPLC.uiActLightLevelPct;

	//calculate BallastOnHours
	fbBallastOnHours(
		bEnableHourCount	:= bEnableHourCount,
		bPauseCount			:= fbLys.fbLightCtrl.bOffZone1,
		uiOnHours			:= uiBallastOnHours_MB,			//OnHours is updated here
		byOverflowCount		:= byOnHoursOverflowCount);


//Manage data for read/write for both PLC and MB registers
fbWriteSPLuxLevel(	nMaxValOut	:= uiMaxLuxLevel,
					nValIn1		:= uiSPLuxLevel_MB,		//nValIn1 takes priotity in case of download or restart
					nValIn2		:= stRoomDataPLC.uiSpLuxLevel,
					nValOut		=> uiLuxOn
				);


fbWritePirDelayTIme(	nMaxValOut	:= uiMaxPirOffMinutes,
						nValIn1		:= uiPirOffDelayTime_MB,		//nValIn1 takes priotity in case of download or restart
						nValIn2		:= stRoomDataPLC.uiPirOffDelayTime,
						nValOut		=> uiPirOffMinutes
					);
					

//Convert read/write modbus data to appropriate datatypes in PLC
fLuxOn	:= TO_REAL(uiLuxOn);			
tPIROff	:= TO_TIME(uiPirOffMinutes*udTimeScaling); //Time conversion defaults to ms

fLuxDim	:= TO_REAL(stRoomDataPLC.uiSpDimLuxLevel);			
tPIRDim	:= TO_TIME(stRoomDataPLC.uiPirDimDelayTime*udTimeScaling); //Time conversion defaults to ms
END_ACTION

ACTION A_Sensor:

fbSensor.ipCommunication := P_DALI_Background.arrfbKL6821Communication[Sesnor_DALI_LINE_NUM];

fbSensor(
	arrShrtAdr:= arrSensorAddr,
	bInitialize:= bInitialize, 
	DALI_LINE_NUM:= Sesnor_DALI_LINE_NUM, 
 	//bCancelHoldTimerOccupancy:= bCancelHoldTimerOccupancy, 
	stSensorSetup := stDaliSensorSetup,
	arrInitErr=> arrInitErr, 
	arrInitDone=> arrInitDone,
	stPirSensorData:= stPirSensorData, 
	arrSensorScales:= arrSensorScales);
END_ACTION

END_PROGRAM

// ---- POUs/Alle_Rum/Rum_Med_DALI_Pir/Rum_1_118/P_Rum_1_118.TcPOU
PROGRAM P_Rum_1_118
VAR
//Light

	fbLys		: FB_Light_Type_A;
	
	stDaliSetup	: SH_Light.ST_DALI_RoomSetup := (		byShrtAdr_Prim := 17, 
														byGrpAdr_Prim := 3, 
														eMod_Prim := E_DALIAddressType.Group, 
														//byShrtAdr_Sec := 1, 
														//byGrpAdr_Sec := 1, 
														//eMod_Sec := E_DALIAddressType.Short, 
														//byShrtAdr_Supl := 1, 
														DALI_LINE_NUM_PRIM := 1, 
														DALI_LINE_NUM_SEC := 0, 
														DALI_LINE_NUM_SUPL := 0);
	stLiveData				: SH_Light.ST_LiveData;
	//stLiveData AT %MB22	: SH_Light.ST_LiveData;
    bRunTuning					: BOOL;
	bTopButtonZone1				: BOOL;
	bTopButtonZone1_Visu		: BOOL;
	bBottomButtonZone1			: BOOL;
	bBottomButtonZone1_Visu	    : BOOL;
	bButtonZone2				: BOOL;
	bNeighborRoomsPir		    : BOOL;
	fLuxOn				     	: REAL;
	fLuxDim						: REAL;
	tPIRDim						: TIME;
	tPIROff						: TIME;
	fOffsetSec					: REAL := 20;
	bOccupiedRoom			    : BOOL;


// Sensor Settings	
	fbSensor					: SH_Light.FB_NIKO_P46xx_2Pcs;
	//fbSensor					: SH_Light.FB_NIKO_P46xx_2Pcs;
	//bySensorAddr				: BYTE := 3;
	arrSensorAddr				: ARRAY[1..2] OF BYTE := [5,6];
	bInitialize					: BOOL := TRUE;
	stDaliSensorSetup			: ST_DALI_NIKOP46SetupData;
	//bInitErr				: BOOL;
	//bInitDone				: BOOL;
	arrInitErr					: ARRAY [1..2] OF BOOL;
	arrInitDone					: ARRAY [1..2] OF BOOL;
	arrSensorScales				: ARRAY [1..10] OF SH_Light.ST_DALI_SensorScaleMode := [	(fMeassureMaxSensor := fMeassure_Zone4, fReadMaxSensor := fRead_Zone4),
																							(fMeassureMaxSensor := fMeassure_Zone4, fReadMaxSensor := fRead_Zone4),
																						8(())];
	bCancelHoldTimerOccupancy	: BOOL;
(*	eEventPriorityOccupancy		: E_DALIEventPriority := E_DALIEVENTPRIORITY.Middle;
	nHoldTimerOccupancy			: WORD := 5; // Value in s. 	
	nReportTimerOccupancy		: BYTE := 120; // Value in s, Preset manufacturer value
	nDeadtimeTimerOccupancy		: WORD := 100; // Value in ms, Predefined Value of DALI Standard
	bCancelHoldTimerOccupancy	: BOOL;
	nSensitivityOccupancy		: BYTE:= 3; //setting Sensivity (0..4) 0 (Off), 1 (Min), 2(Low), 3(High) and 4 (Max)

	bEnableLuxEvent				: BOOL;
	eEventPriorityBrightness	: E_DALIEventPriority := E_DALIEVENTPRIORITY.Middle;
	nDeadtimeTimerBrightness	: WORD := 1500; // Value in ms, Predefined Value of DALI Standard
	nHysteresisBrightness		: BYTE := 2; // Value in %
	nHysteresisMinBrightness	: BYTE := 10; // Absolute Value, depending on the manufacturer specific resolution
	nReportTimerBrightness		: BYTE := 120; // Value in s, Preset manufacturer value
*)


	//ModbusComm setup
	
	fbWriteSPLuxLevel			: SH_Light.FB_TwoVal_SelectOne_RTrigChange;
	fbWritePirDelayTIme		: SH_Light.FB_TwoVal_SelectOne_RTrigChange;
	stRoomDataPLC				: SH_Light.ST_RoomDataPLC	:=	(
																	uiPirOffDelayTime	:= 30,
																	uiSpLuxLevel		:= 500,
																	uiPirDimDelayTime	:= 15,
																	uiSpDimLuxLevel		:= 200);
																	
	fbBallastOnHours				: SH_Light.FB_CountOnHours;
	bEnableHourCount			: BOOL := TRUE;
	
	//Non-persistent modbus data
	bPirActive_MB					AT %MX80.0	: BOOL;				//bPirLys i gammel kode
	uiActLuxLevel_MB			    AT %MB84	: UINT;				//intHMIAktueltLux i gammel kode
	uiActLightLevelPct_MB	        AT %MB88	: UINT;				//intDALI_Gruppe1_Lysniveau i gammel kode
	
	//For Conversion
	uiPirOffMinutes						: UINT;
	udTimeScaling						: UDINT := 60000;
	uiLuxOn								: UINT;
	
	//max values checks
	uiMaxLuxLevel						: UINT := 1023;
	uiMaxPirOffMinutes				    : UINT := 180;

END_VAR

VAR CONSTANT
	Sesnor_DALI_LINE_NUM: BYTE := 2;
	DALI_LINE_NUM_LIGHT: BYTE := 1;
	DALI_LINE_NUM_PENDANTS	            : BYTE := 0; //0=ingen pendler	
	arrSensitivityOccupancy				: ARRAY[1..3] OF BYTE := [4,4,4]; //sensitivitet for sensor

END_VAR
VAR PERSISTENT
	stPirSensorData: SH_Light.ST_DALI_Sensor;
	stTuneData: SH_Light.ST_TuneData_EX;
	
	uiPirOffDelayTime_MB	AT %MB82	: UINT;				//ntHMI_Pir_SetValue i gammel kode
	uiSPLuxLevel_MB			AT %MB86	: UINT;				//intHMI_Lux_SetValue i gammel kode
	uiBallastOnHours_MB		AT %MB90	: UINT;				//dintHMILysbraendtimer1 i gammel kode
	byOnHoursOverflowCount				: BYTE;   

END_VAR

A_Buttons();
A_LightCtrl();
A_Sensor();
A_Modbuscomm();

ACTION A_Buttons:
bTopButtonZone1		:= GVL_EnOcean.strEnOceanSwitch_Rum_1_118.bT1_ON OR bTopButtonZone1_Visu;
bBottomButtonZone1	:= GVL_EnOcean.strEnOceanSwitch_Rum_1_118.bT1_OFF OR bBottomButtonZone1_Visu;
END_ACTION

ACTION A_LightCtrl:

fbLys(
	nZoneID:= 1, 
	bButtonZone1:= bTopButtonZone1,
	bBottomButtonZone1 := bBottomButtonZone1, 
	bButtonZone2:= bButtonZone2, 
	fLuxOn:= fLuxOn, 
	fLuxDim:= fLuxDim, 
	tPIRDim:= tPIRDim, 
	tPIROff:= tPIROff, 
	fOffsetSec:= fOffsetSec, 
	bReInit:= , 
	stDaliSetup:= stDaliSetup, 
	ipCommunication_Prim:= P_DALI_Background.arrfbKL6821Communication[DALI_LINE_NUM_LIGHT], 
	//ipCommunication_Sec:= P_DALI_Background.arrfbKL6821Communication[DALI_LINE_NUM_LIGHT], 
	//ipCommunication_Supl:= P_DALI_Background.arrfbKL6821Communication[DALI_LINE_NUM_LIGHT], 
	fMinOutputPowerLevelRoom:= 15, 
	fMaxOutputPowerLevelRoom:= 100, 
	nCycleTimeInMS:= SH_Light.DALI_Param.nPlcTaskCycleTimeInMS*nDimCmdCycleTimeFactor  , 
	bRunTuning:= bRunTuning, 
	bOccupiedRoom=> bOccupiedRoom, 
	bError_Prim=> , 
	nError_Prim=> , 
	stTuneData:=stTuneData , 
	stPirSensorData:= stPirSensorData, 
	stLiveData:= stLiveData);
END_ACTION

ACTION A_ModbusComm:
//Manage data for modbus communication

//Manage data for read-only in PLC
stRoomDataPLC.bPirActive			:= stPirSensorData.bPrc;
stRoomDataPLC.uiActLuxLevel			:= TO_UINT(TRUNC(stPirSensorData.fBrightness));
stRoomDataPLC.uiActLightLevelPct	:= TO_UINT(TRUNC(fbLys.fbBallast.fActlLgtLvl_Prim));
		//stRoomDataPLC.uiActLightLevelPct	:= TO_UINT(TRUNC(fbLys.fbBallast.fActlLgtLvl_Prim)); //if only one group light control
stRoomDataPLC.uiBallastOnHours		:= uiBallastOnHours_MB; //The calculation for BallastOnHours is stored directly to the MB register below


//Assign data for read-only to MB registers
bPirActive_MB			:= stRoomDataPLC.bPirActive;
uiActLuxLevel_MB		:= stRoomDataPLC.uiActLuxLevel;
uiActLightLevelPct_MB	:= stRoomDataPLC.uiActLightLevelPct;

	//calculate BallastOnHours
	fbBallastOnHours(
		bEnableHourCount	:= bEnableHourCount,
		bPauseCount			:= fbLys.fbLightCtrl.bOffZone1,
		uiOnHours			:= uiBallastOnHours_MB,			//OnHours is updated here
		byOverflowCount		:= byOnHoursOverflowCount);


//Manage data for read/write for both PLC and MB registers
fbWriteSPLuxLevel(	nMaxValOut	:= uiMaxLuxLevel,
					nValIn1		:= uiSPLuxLevel_MB,		//nValIn1 takes priotity in case of download or restart
					nValIn2		:= stRoomDataPLC.uiSpLuxLevel,
					nValOut		=> uiLuxOn
				);


fbWritePirDelayTIme(	nMaxValOut	:= uiMaxPirOffMinutes,
						nValIn1		:= uiPirOffDelayTime_MB,		//nValIn1 takes priotity in case of download or restart
						nValIn2		:= stRoomDataPLC.uiPirOffDelayTime,
						nValOut		=> uiPirOffMinutes
					);
					

//Convert read/write modbus data to appropriate datatypes in PLC
fLuxOn	:= TO_REAL(uiLuxOn);			
tPIROff	:= TO_TIME(uiPirOffMinutes*udTimeScaling); //Time conversion defaults to ms

fLuxDim	:= TO_REAL(stRoomDataPLC.uiSpDimLuxLevel);			
tPIRDim	:= TO_TIME(stRoomDataPLC.uiPirDimDelayTime*udTimeScaling); //Time conversion defaults to ms
END_ACTION

ACTION A_Sensor:

fbSensor.ipCommunication := P_DALI_Background.arrfbKL6821Communication[Sesnor_DALI_LINE_NUM];

fbSensor(
	arrShrtAdr:= arrSensorAddr,
	bInitialize:= bInitialize, 
	DALI_LINE_NUM:= Sesnor_DALI_LINE_NUM, 
 	//bCancelHoldTimerOccupancy:= bCancelHoldTimerOccupancy, 
	stSensorSetup := stDaliSensorSetup,
	arrInitErr=> arrInitErr, 
	arrInitDone=> arrInitDone,
	stPirSensorData:= stPirSensorData, 
	arrSensorScales:= arrSensorScales);
END_ACTION

END_PROGRAM

// ---- POUs/Alle_Rum/Gange/P_Gang_1_111A/P_Gang_1_111A.TcPOU
PROGRAM P_Gang_1_111A
VAR
//Light

	fbLys		: FB_Light_Type_B;
	
	stDaliSetup	: SH_Light.ST_DALI_RoomSetup := (		byShrtAdr_Prim := 47, 
														byGrpAdr_Prim := 6, 
														eMod_Prim := E_DALIAddressType.Group, 
														//byShrtAdr_Sec := 1, 
														//byGrpAdr_Sec := 1, 
														//eMod_Sec := E_DALIAddressType.Short, 
														//byShrtAdr_Supl := 1, 
														DALI_LINE_NUM_PRIM := 2, 
														DALI_LINE_NUM_SEC := 0, 
														DALI_LINE_NUM_SUPL := 0);
														
	stLiveData				: SH_Light.ST_LiveData;
	bRunTuning					: BOOL;
	
	bTopButtonZone1				: BOOL;
	bTopButtonZone1_Visu		: BOOL;
	bBottomButtonZone1			: BOOL;
	bBottomButtonZone1_Visu	    : BOOL;
	bButtonZone2				: BOOL;
	bNeighborRoomsPir		    : BOOL;
	fLuxOn				     	: REAL;
	fLuxDim						: REAL;
	tPIRDim						: TIME;
	tPIROff						: TIME;
	fOffsetSec					: REAL := 20;
	bOccupiedRoom			    : BOOL;



// Sensor Settings	
	fbSensor					: SH_Light.FB_NIKO_P46xx_1Pcs;
	//fbSensor					: SH_Light.FB_NIKO_P46xx_2Pcs;
	bySensorAddr				: BYTE := 11;                           //ved en sensor
	//arrSensorAddr				: ARRAY[1..2] OF BYTE := [7,8];         // Ved flere
	bInitialize					: BOOL := TRUE;
	stDaliSensorSetup			: ST_DALI_NIKOP46SetupData := (
																nSensitivityPIRSegmentA := arrSensitivityOccupancy[1],
																nSensitivityPIRSegmentB := arrSensitivityOccupancy[2],
																nSensitivityPIRSegmentC := arrSensitivityOccupancy[3]);

	bInitErr				: BOOL;                                     //ved en sensor
	bInitDone				: BOOL;                                     //Ved en sensor 
	//arrInitErr					: ARRAY [1..2] OF BOOL;             // Ved flere 
	//arrInitDone					: ARRAY [1..2] OF BOOL;             //Ved flere
	arrSensorScales				: ARRAY [1..10] OF SH_Light.ST_DALI_SensorScaleMode := [	(fMeassureMaxSensor := fMeassure_Zone10, fReadMaxSensor := fRead_Zone10),
																						9(())];
	bCancelHoldTimerOccupancy	: BOOL;
(*	eEventPriorityOccupancy		: E_DALIEventPriority := E_DALIEVENTPRIORITY.Middle;
	nHoldTimerOccupancy			: WORD := 5; // Value in s. 	
	nReportTimerOccupancy		: BYTE := 120; // Value in s, Preset manufacturer value
	nDeadtimeTimerOccupancy		: WORD := 100; // Value in ms, Predefined Value of DALI Standard
	bCancelHoldTimerOccupancy	: BOOL;
	nSensitivityOccupancy		: BYTE:= 3; //setting Sensivity (0..4) 0 (Off), 1 (Min), 2(Low), 3(High) and 4 (Max)

	bEnableLuxEvent				: BOOL;
	eEventPriorityBrightness	: E_DALIEventPriority := E_DALIEVENTPRIORITY.Middle;
	nDeadtimeTimerBrightness	: WORD := 1500; // Value in ms, Predefined Value of DALI Standard
	nHysteresisBrightness		: BYTE := 2; // Value in %
	nHysteresisMinBrightness	: BYTE := 10; // Absolute Value, depending on the manufacturer specific resolution
	nReportTimerBrightness		: BYTE := 120; // Value in s, Preset manufacturer value
*)

	//ModbusComm setup
	
	fbWriteSPLuxLevel			: SH_Light.FB_TwoVal_SelectOne_RTrigChange;
	fbWritePirDelayTIme		: SH_Light.FB_TwoVal_SelectOne_RTrigChange;
	stRoomDataPLC				: SH_Light.ST_RoomDataPLC	:=	(
																	uiPirOffDelayTime	:= 30,
																	uiSpLuxLevel		:= 500,
																	uiPirDimDelayTime	:= 15,
																	uiSpDimLuxLevel		:= 200);
																	
	fbBallastOnHours				: SH_Light.FB_CountOnHours;
	bEnableHourCount			: BOOL := TRUE;
	
	//Non-persistent modbus data
	bPirActive_MB					AT %MX524.0	: BOOL;				//bPirLys i gammel kode
	uiActLuxLevel_MB			    AT %MB528	: UINT;				//intHMIAktueltLux i gammel kode
	uiActLightLevelPct_MB	        AT %MB532	: UINT;				//intDALI_Gruppe1_Lysniveau i gammel kode
	
	//For Conversion
	uiPirOffMinutes						: UINT;
	udTimeScaling						: UDINT := 60000;
	uiLuxOn								: UINT;
	
	//max values checks
	uiMaxLuxLevel						: UINT := 1023;
	uiMaxPirOffMinutes				    : UINT := 180;

	
END_VAR

VAR CONSTANT
	Sesnor_DALI_LINE_NUM: INT := 2;
	DALI_LINE_NUM_LIGHT: INT := 2;
	DALI_LINE_NUM_PENDANTS	            : BYTE := 0; //0=ingen pendler	
	arrSensitivityOccupancy				: ARRAY[1..3] OF BYTE := [4,4,4]; //sensitivitet for sensor

END_VAR
VAR PERSISTENT
	stPirSensorData: SH_Light.ST_DALI_Sensor;
	stTuneData: SH_Light.ST_TuneData_EX;
	
	uiPirOffDelayTime_MB	AT %MB526	: UINT;				//ntHMI_Pir_SetValue i gammel kode
	uiSPLuxLevel_MB			AT %MB530	: UINT;				//intHMI_Lux_SetValue i gammel kode
	uiBallastOnHours_MB		AT %MB534	: UINT;				//dintHMILysbraendtimer1 i gammel kode
	byOnHoursOverflowCount				: BYTE;   
END_VAR

A_Buttons();
A_LightCtrl();
A_Sensor();
A_modbuscomm();

ACTION A_Buttons:
bTopButtonZone1		:= bTopButtonZone1_Visu;
bBottomButtonZone1	:= bBottomButtonZone1_Visu;
END_ACTION

ACTION A_LightCtrl:
bNeighborRoomsPir	:= P_gang_1_108.stPirSensorData.bPrc OR P_Rum_1_111E.stPirSensorData.bPrc OR P_Rum_1_111C.stPirSensorData.bPrc OR P_Rum_1_111D.stPirSensorData.bPrc ; ///husk 111C og D
fbLys( 
	nZoneID:= 1, 
	bButtonZone1:= bTopButtonZone1,
	bBottomButtonZone1 := bBottomButtonZone1, 
	//bButtonZone2:= bButtonZone2,
	bNeighborRoomsPir	:=	bNeighborRoomsPir,
	fLuxOn:= fLuxOn, 
	fLuxDim:= fLuxDim, 
	tPIRDim:= tPIRDim, 
	tPIROff:= tPIROff, 
	fOffsetSec:= fOffsetSec, 
	bReInit:= , 
	stDaliSetup:= stDaliSetup, 
	ipCommunication_Prim:= P_DALI_Background.arrfbKL6821Communication[DALI_LINE_NUM_LIGHT], 
	//ipCommunication_Sec:= P_DALI_Background.arrfbKL6821Communication[DALI_LINE_NUM_LIGHT], 
	//ipCommunication_Supl:= P_DALI_Background.arrfbKL6821Communication[DALI_LINE_NUM_LIGHT], 
	fMinOutputPowerLevelRoom:= 15, 
	fMaxOutputPowerLevelRoom:= 100, 
	nCycleTimeInMS:= SH_Light.DALI_Param.nPlcTaskCycleTimeInMS*nDimCmdCycleTimeFactor, 
	bRunTuning:= bRunTuning, 
	bOccupiedRoom=> bOccupiedRoom, 
	bError_Prim=> , 
	nError_Prim=> , 
	stTuneData:=stTuneData , 
	stPirSensorData:= stPirSensorData, 
	stLiveData:= stLiveData);
END_ACTION

ACTION A_ModbusComm:
//Manage data for modbus communication

//Manage data for read-only in PLC
stRoomDataPLC.bPirActive			:= stPirSensorData.bPrc;
stRoomDataPLC.uiActLuxLevel			:= TO_UINT(TRUNC(stPirSensorData.fBrightness));
stRoomDataPLC.uiActLightLevelPct	:= TO_UINT(TRUNC(fbLys.fbBallast.fActlLgtLvl_Prim));
		//stRoomDataPLC.uiActLightLevelPct	:= TO_UINT(TRUNC(fbLys.fbBallast.fActlLgtLvl_Prim)); //if only one group light control
stRoomDataPLC.uiBallastOnHours		:= uiBallastOnHours_MB; //The calculation for BallastOnHours is stored directly to the MB register below


//Assign data for read-only to MB registers
bPirActive_MB			:= stRoomDataPLC.bPirActive;
uiActLuxLevel_MB		:= stRoomDataPLC.uiActLuxLevel;
uiActLightLevelPct_MB	:= stRoomDataPLC.uiActLightLevelPct;

	//calculate BallastOnHours
	fbBallastOnHours(
		bEnableHourCount	:= bEnableHourCount,
		bPauseCount			:= fbLys.fbLightCtrl.bOffZone1,
		uiOnHours			:= uiBallastOnHours_MB,			//OnHours is updated here
		byOverflowCount		:= byOnHoursOverflowCount);


//Manage data for read/write for both PLC and MB registers
fbWriteSPLuxLevel(	nMaxValOut	:= uiMaxLuxLevel,
					nValIn1		:= uiSPLuxLevel_MB,		//nValIn1 takes priotity in case of download or restart
					nValIn2		:= stRoomDataPLC.uiSpLuxLevel,
					nValOut		=> uiLuxOn
				);


fbWritePirDelayTIme(	nMaxValOut	:= uiMaxPirOffMinutes,
						nValIn1		:= uiPirOffDelayTime_MB,		//nValIn1 takes priotity in case of download or restart
						nValIn2		:= stRoomDataPLC.uiPirOffDelayTime,
						nValOut		=> uiPirOffMinutes
					);
					

//Convert read/write modbus data to appropriate datatypes in PLC
fLuxOn	:= TO_REAL(uiLuxOn);			
tPIROff	:= TO_TIME(uiPirOffMinutes*udTimeScaling); //Time conversion defaults to ms

fLuxDim	:= TO_REAL(stRoomDataPLC.uiSpDimLuxLevel);			
tPIRDim	:= TO_TIME(stRoomDataPLC.uiPirDimDelayTime*udTimeScaling); //Time conversion defaults to ms
END_ACTION

ACTION A_Sensor:

fbSensor.ipCommunication := P_DALI_Background.arrfbKL6821Communication[Sesnor_DALI_LINE_NUM];

fbSensor(
	byShrtAdr:= bySensorAddr,
	bInitialize:= bInitialize, 
	DALI_LINE_NUM:= Sesnor_DALI_LINE_NUM, 
 	//bCancelHoldTimerOccupancy:= bCancelHoldTimerOccupancy, 
	stSensorSetup := stDaliSensorSetup,
	bInitErr=> bInitErr, 
	bInitDone=> bInitDone,
	stPirSensorData:= stPirSensorData, 
	arrSensorScales:= arrSensorScales);
END_ACTION

END_PROGRAM

// ---- POUs/Alle_Rum/Rum_Med_DALI_Pir/Rum_1_111E/P_Rum_1_111E.TcPOU
PROGRAM P_Rum_1_111E
VAR
//Light

	fbLys		: FB_Light_Type_A;
	
	stDaliSetup	: SH_Light.ST_DALI_RoomSetup := (		byShrtAdr_Prim := 1, 
														byGrpAdr_Prim := 1, 
														eMod_Prim := E_DALIAddressType.Group, 
														//byShrtAdr_Sec := 1, 
														//byGrpAdr_Sec := 1, 
														//eMod_Sec := E_DALIAddressType.Short, 
														//byShrtAdr_Supl := 1, 
														DALI_LINE_NUM_PRIM := 1, 
														DALI_LINE_NUM_SEC := 0, 
														DALI_LINE_NUM_SUPL := 0);
	stLiveData				: SH_Light.ST_LiveData;
	//stLiveData AT %MB22	: SH_Light.ST_LiveData;
	bRunTuning					: BOOL;
	
	bTopButtonZone1				: BOOL;
	bTopButtonZone1_Visu		: BOOL;
	bBottomButtonZone1			: BOOL;
	bBottomButtonZone1_Visu	    : BOOL;
	bButtonZone2				: BOOL;
	bNeighborRoomsPir		    : BOOL;
	fLuxOn				     	: REAL;
	fLuxDim						: REAL;
	tPIRDim						: TIME;
	tPIROff						: TIME;
	fOffsetSec					: REAL := 20;
	bOccupiedRoom			    : BOOL;


// Sensor Settings	
	fbSensor					: SH_Light.FB_NIKO_P46xx_1Pcs;
	//fbSensor					: SH_Light.FB_NIKO_P46xx_2Pcs;
	bySensorAddr				: BYTE := 1;
	//arrSensorAddr				: ARRAY[1..2] OF BOOL;
	bInitialize					: BOOL := TRUE;
	stDaliSensorSetup			: ST_DALI_NIKOP46SetupData := (
																nSensitivityPIRSegmentA := arrSensitivityOccupancy[1],
																nSensitivityPIRSegmentB := arrSensitivityOccupancy[2],
																nSensitivityPIRSegmentC := arrSensitivityOccupancy[3]);

	bInitErr				: BOOL;
	bInitDone				: BOOL;
	//arrInitErr					: ARRAY [1..2] OF BOOL;
	//arrInitDone					: ARRAY [1..2] OF BOOL;
	arrSensorScales				: ARRAY [1..10] OF SH_Light.ST_DALI_SensorScaleMode := [	(fMeassureMaxSensor := fMeassure_Zone3, fReadMaxSensor := fRead_Zone3),
																						9(())];
	bCancelHoldTimerOccupancy	: BOOL;
(*	eEventPriorityOccupancy		: E_DALIEventPriority := E_DALIEVENTPRIORITY.Middle;
	nHoldTimerOccupancy			: WORD := 5; // Value in s. 	
	nReportTimerOccupancy		: BYTE := 120; // Value in s, Preset manufacturer value
	nDeadtimeTimerOccupancy		: WORD := 100; // Value in ms, Predefined Value of DALI Standard
	bCancelHoldTimerOccupancy	: BOOL;
	nSensitivityOccupancy		: BYTE:= 3; //setting Sensivity (0..4) 0 (Off), 1 (Min), 2(Low), 3(High) and 4 (Max)

	bEnableLuxEvent				: BOOL;
	eEventPriorityBrightness	: E_DALIEventPriority := E_DALIEVENTPRIORITY.Middle;
	nDeadtimeTimerBrightness	: WORD := 1500; // Value in ms, Predefined Value of DALI Standard
	nHysteresisBrightness		: BYTE := 2; // Value in %
	nHysteresisMinBrightness	: BYTE := 10; // Absolute Value, depending on the manufacturer specific resolution
	nReportTimerBrightness		: BYTE := 120; // Value in s, Preset manufacturer value
*)

	//ModbusComm setup
	
	fbWriteSPLuxLevel			: SH_Light.FB_TwoVal_SelectOne_RTrigChange;
	fbWritePirDelayTIme		: SH_Light.FB_TwoVal_SelectOne_RTrigChange;
	stRoomDataPLC				: SH_Light.ST_RoomDataPLC	:=	(
																	uiPirOffDelayTime	:= 30,
																	uiSpLuxLevel		:= 500,
																	uiPirDimDelayTime	:= 15,
																	uiSpDimLuxLevel		:= 200);
																	
	fbBallastOnHours				: SH_Light.FB_CountOnHours;
	bEnableHourCount			: BOOL := TRUE;
	
	//Non-persistent modbus data
	bPirActive_MB					AT %MX32.0	: BOOL;				//bPirLys i gammel kode
	uiActLuxLevel_MB			    AT %MB36	: UINT;				//intHMIAktueltLux i gammel kode
	uiActLightLevelPct_MB	        AT %MB40	: UINT;				//intDALI_Gruppe1_Lysniveau i gammel kode
	
	//For Conversion
	uiPirOffMinutes						: UINT;
	udTimeScaling						: UDINT := 60000;
	uiLuxOn								: UINT;
	
	//max values checks
	uiMaxLuxLevel						: UINT := 1023;
	uiMaxPirOffMinutes				    : UINT := 180;

END_VAR

VAR CONSTANT
	Sesnor_DALI_LINE_NUM: BYTE := 2;
	DALI_LINE_NUM_LIGHT: BYTE := 1;
		DALI_LINE_NUM_PENDANTS	            : BYTE := 0; //0=ingen pendler	
	arrSensitivityOccupancy				: ARRAY[1..3] OF BYTE := [4,4,4]; //sensitivitet for sensor

END_VAR
VAR PERSISTENT
	stPirSensorData: SH_Light.ST_DALI_Sensor;
	stTuneData: SH_Light.ST_TuneData_EX;
	
	uiPirOffDelayTime_MB	AT%MB34		: UINT;				//ntHMI_Pir_SetValue i gammel kode
	uiSPLuxLevel_MB			AT%MB38		: UINT;				//intHMI_Lux_SetValue i gammel kode
	uiBallastOnHours_MB		AT%MB42		: UINT;				//dintHMILysbraendtimer1 i gammel kode
 	byOnHoursOverflowCount				: BYTE;   

END_VAR

A_Buttons();
A_LightCtrl();
A_ModbusComm();
A_Sensor();

ACTION A_Buttons:
bTopButtonZone1		:= GVL_EnOcean.strEnOceanSwitch_Rum_1_111E.bT2_ON OR bTopButtonZone1_Visu;
bBottomButtonZone1	:= GVL_EnOcean.strEnOceanSwitch_Rum_1_111E.bT2_OFF OR bBottomButtonZone1_Visu;
END_ACTION

ACTION A_LightCtrl:

fbLys(
	nZoneID:= 1, 
	bButtonZone1:= bTopButtonZone1,
	bBottomButtonZone1 := bBottomButtonZone1, 
	//bButtonZone2:= bButtonZone2, 
	fLuxOn:= fLuxOn, 
	fLuxDim:= fLuxDim, 
	tPIRDim:= tPIRDim, 
	tPIROff:= tPIROff, 
	fOffsetSec:= fOffsetSec, 
	bReInit:= , 
	stDaliSetup:= stDaliSetup, 
	ipCommunication_Prim:= P_DALI_Background.arrfbKL6821Communication[DALI_LINE_NUM_LIGHT], 
	//ipCommunication_Sec:= P_DALI_Background.arrfbKL6821Communication[DALI_LINE_NUM_LIGHT], 
	//ipCommunication_Supl:= P_DALI_Background.arrfbKL6821Communication[DALI_LINE_NUM_LIGHT], 
	fMinOutputPowerLevelRoom:= 15, 
	fMaxOutputPowerLevelRoom:= 100, 
	nCycleTimeInMS:=  SH_Light.DALI_Param.nPlcTaskCycleTimeInMS*nDimCmdCycleTimeFactor  , 
	bRunTuning:= bRunTuning, 
	bOccupiedRoom=> bOccupiedRoom, 
	bError_Prim=> , 
	nError_Prim=> , 
	stTuneData:=stTuneData , 
	stPirSensorData:= stPirSensorData, 
	stLiveData:= stLiveData);
END_ACTION

ACTION A_ModbusComm:
//Manage data for modbus communication

//Manage data for read-only in PLC
stRoomDataPLC.bPirActive			:= stPirSensorData.bPrc;
stRoomDataPLC.uiActLuxLevel			:= TO_UINT(TRUNC(stPirSensorData.fBrightness));
stRoomDataPLC.uiActLightLevelPct	:= TO_UINT(TRUNC(fbLys.fbBallast.fActlLgtLvl_Prim));
		//stRoomDataPLC.uiActLightLevelPct	:= TO_UINT(TRUNC(fbLys.fbBallast.fActlLgtLvl_Prim)); //if only one group light control
stRoomDataPLC.uiBallastOnHours		:= uiBallastOnHours_MB; //The calculation for BallastOnHours is stored directly to the MB register below


//Assign data for read-only to MB registers
bPirActive_MB			:= stRoomDataPLC.bPirActive;
uiActLuxLevel_MB		:= stRoomDataPLC.uiActLuxLevel;
uiActLightLevelPct_MB	:= stRoomDataPLC.uiActLightLevelPct;

	//calculate BallastOnHours
	fbBallastOnHours(
		bEnableHourCount	:= bEnableHourCount,
		bPauseCount			:= fbLys.fbLightCtrl.bOffZone1,
		uiOnHours			:= uiBallastOnHours_MB,			//OnHours is updated here
		byOverflowCount		:= byOnHoursOverflowCount);


//Manage data for read/write for both PLC and MB registers
fbWriteSPLuxLevel(	nMaxValOut	:= uiMaxLuxLevel,
					nValIn1		:= uiSPLuxLevel_MB,		//nValIn1 takes priotity in case of download or restart
					nValIn2		:= stRoomDataPLC.uiSpLuxLevel,
					nValOut		=> uiLuxOn
				);


fbWritePirDelayTIme(	nMaxValOut	:= uiMaxPirOffMinutes,
						nValIn1		:= uiPirOffDelayTime_MB,		//nValIn1 takes priotity in case of download or restart
						nValIn2		:= stRoomDataPLC.uiPirOffDelayTime,
						nValOut		=> uiPirOffMinutes
					);
					

//Convert read/write modbus data to appropriate datatypes in PLC
fLuxOn	:= TO_REAL(uiLuxOn);			
tPIROff	:= TO_TIME(uiPirOffMinutes*udTimeScaling); //Time conversion defaults to ms

fLuxDim	:= TO_REAL(stRoomDataPLC.uiSpDimLuxLevel);			
tPIRDim	:= TO_TIME(stRoomDataPLC.uiPirDimDelayTime*udTimeScaling); //Time conversion defaults to ms
END_ACTION

ACTION A_Sensor:

fbSensor.ipCommunication := P_DALI_Background.arrfbKL6821Communication[Sesnor_DALI_LINE_NUM];

fbSensor(
	byShrtAdr:= bySensorAddr, 
	bInitialize:= bInitialize, 
	DALI_LINE_NUM:= Sesnor_DALI_LINE_NUM, 
 	//bCancelHoldTimerOccupancy:= bCancelHoldTimerOccupancy, 
	stSensorSetup := stDaliSensorSetup,
	bInitErr=> bInitErr, 
	bInitDone=> bInitDone,
	stPirSensorData:= stPirSensorData, 
	arrSensorScales:= arrSensorScales);
END_ACTION

END_PROGRAM

// ---- POUs/Alle_Rum/Rum_Med_DALI_Pir/Rum_1_111C/P_Rum_1_111C.TcPOU
PROGRAM P_Rum_1_111C
VAR
//Light

	fbLys		: FB_Light_Type_A;
	
	stDaliSetup	: SH_Light.ST_DALI_RoomSetup := (		byShrtAdr_Prim := 50, 
														byGrpAdr_Prim := 7, 
														eMod_Prim := E_DALIAddressType.Group, 
														//byShrtAdr_Sec := 1, 
														//byGrpAdr_Sec := 1, 
														//eMod_Sec := E_DALIAddressType.Short, 
														//byShrtAdr_Supl := 1, 
														DALI_LINE_NUM_PRIM := 2, 
														DALI_LINE_NUM_SEC := 0, 
														DALI_LINE_NUM_SUPL := 0);
	stLiveData				: SH_Light.ST_LiveData;
	//stLiveData AT %MB22	: SH_Light.ST_LiveData;
		bRunTuning					: BOOL;
	
	bTopButtonZone1				: BOOL;
	bTopButtonZone1_Visu		: BOOL;
	bBottomButtonZone1			: BOOL;
	bBottomButtonZone1_Visu	    : BOOL;
	bButtonZone2				: BOOL;
	bNeighborRoomsPir		    : BOOL;
	fLuxOn				     	: REAL;
	fLuxDim						: REAL;
	tPIRDim						: TIME;
	tPIROff						: TIME;
	fOffsetSec					: REAL := 20;
	bOccupiedRoom			    : BOOL;


// Sensor Settings	
	fbSensor					: SH_Light.FB_NIKO_P46xx_1Pcs;
	//fbSensor					: SH_Light.FB_NIKO_P46xx_2Pcs;
	bySensorAddr				: BYTE := 12;
	//arrSensorAddr				: ARRAY[1..2] OF BOOL;
	bInitialize					: BOOL := TRUE;
	stDaliSensorSetup			: ST_DALI_NIKOP46SetupData := (
																nSensitivityPIRSegmentA := arrSensitivityOccupancy[1],
																nSensitivityPIRSegmentB := arrSensitivityOccupancy[2],
																nSensitivityPIRSegmentC := arrSensitivityOccupancy[3]);

	bInitErr				: BOOL;
	bInitDone				: BOOL;
	//arrInitErr					: ARRAY [1..2] OF BOOL;
	//arrInitDone					: ARRAY [1..2] OF BOOL;
	arrSensorScales				: ARRAY [1..10] OF SH_Light.ST_DALI_SensorScaleMode := [	(fMeassureMaxSensor := fMeassure_Zone10, fReadMaxSensor := fRead_Zone10), 
																						9(())];
	bCancelHoldTimerOccupancy	: BOOL;
(*	eEventPriorityOccupancy		: E_DALIEventPriority := E_DALIEVENTPRIORITY.Middle;
	nHoldTimerOccupancy			: WORD := 5; // Value in s. 	
	nReportTimerOccupancy		: BYTE := 120; // Value in s, Preset manufacturer value
	nDeadtimeTimerOccupancy		: WORD := 100; // Value in ms, Predefined Value of DALI Standard
	bCancelHoldTimerOccupancy	: BOOL;
	nSensitivityOccupancy		: BYTE:= 3; //setting Sensivity (0..4) 0 (Off), 1 (Min), 2(Low), 3(High) and 4 (Max)

	bEnableLuxEvent				: BOOL;
	eEventPriorityBrightness	: E_DALIEventPriority := E_DALIEVENTPRIORITY.Middle;
	nDeadtimeTimerBrightness	: WORD := 1500; // Value in ms, Predefined Value of DALI Standard
	nHysteresisBrightness		: BYTE := 2; // Value in %
	nHysteresisMinBrightness	: BYTE := 10; // Absolute Value, depending on the manufacturer specific resolution
	nReportTimerBrightness		: BYTE := 120; // Value in s, Preset manufacturer value
*)

	//ModbusComm setup
	
	fbWriteSPLuxLevel			: SH_Light.FB_TwoVal_SelectOne_RTrigChange;
	fbWritePirDelayTIme		: SH_Light.FB_TwoVal_SelectOne_RTrigChange;
	stRoomDataPLC				: SH_Light.ST_RoomDataPLC	:=	(
																	uiPirOffDelayTime	:= 30,
																	uiSpLuxLevel		:= 500,
																	uiPirDimDelayTime	:= 15,
																	uiSpDimLuxLevel		:= 200);
																	
	fbBallastOnHours				: SH_Light.FB_CountOnHours;
	bEnableHourCount			: BOOL := TRUE;
	
	//Non-persistent modbus data
	bPirActive_MB					AT %MX512.0	: BOOL;				//bPirLys i gammel kode
	uiActLuxLevel_MB			    AT %MB516	: UINT;				//intHMIAktueltLux i gammel kode
	uiActLightLevelPct_MB	        AT %MB520	: UINT;				//intDALI_Gruppe1_Lysniveau i gammel kode
	
	//For Conversion
	uiPirOffMinutes						: UINT;
	udTimeScaling						: UDINT := 60000;
	uiLuxOn								: UINT;
	
	//max values checks
	uiMaxLuxLevel						: UINT := 1023;
	uiMaxPirOffMinutes				    : UINT := 180;

END_VAR

VAR CONSTANT
	Sesnor_DALI_LINE_NUM: BYTE := 2;
	DALI_LINE_NUM_LIGHT: BYTE := 2;
	DALI_LINE_NUM_PENDANTS	            : BYTE := 0; //0=ingen pendler	
	arrSensitivityOccupancy				: ARRAY[1..3] OF BYTE := [4,4,4]; //sensitivitet for sensor

END_VAR
VAR PERSISTENT
	stPirSensorData: SH_Light.ST_DALI_Sensor;
	stTuneData: SH_Light.ST_TuneData_EX;
	
	uiPirOffDelayTime_MB	AT %MB514	: UINT;				//ntHMI_Pir_SetValue i gammel kode
	uiSPLuxLevel_MB			AT %MB518	: UINT;				//intHMI_Lux_SetValue i gammel kode
	uiBallastOnHours_MB		AT %MB522	: UINT;				//dintHMILysbraendtimer1 i gammel kode
	byOnHoursOverflowCount				: BYTE;   

END_VAR

A_Buttons();
A_LightCtrl();
A_Sensor();
A_Modbuscomm();

ACTION A_Buttons:
bTopButtonZone1		:= bTopButtonZone1_Visu;
bBottomButtonZone1	:= bBottomButtonZone1_Visu;
END_ACTION

ACTION A_LightCtrl:

fbLys(
	nZoneID:= 1, 
	bButtonZone1:= bTopButtonZone1,
	bBottomButtonZone1 := bBottomButtonZone1, 
	bButtonZone2:= bButtonZone2, 
	fLuxOn:= fLuxOn, 
	fLuxDim:= fLuxDim, 
	tPIRDim:= tPIRDim, 
	tPIROff:= tPIROff, 
	fOffsetSec:= fOffsetSec, 
	bReInit:= , 
	stDaliSetup:= stDaliSetup, 
	ipCommunication_Prim:= P_DALI_Background.arrfbKL6821Communication[DALI_LINE_NUM_LIGHT], 
	//ipCommunication_Sec:= P_DALI_Background.arrfbKL6821Communication[DALI_LINE_NUM_LIGHT], 
	//ipCommunication_Supl:= P_DALI_Background.arrfbKL6821Communication[DALI_LINE_NUM_LIGHT], 
	fMinOutputPowerLevelRoom:= 15, 
	fMaxOutputPowerLevelRoom:= 100, 
	nCycleTimeInMS:= SH_Light.DALI_Param.nPlcTaskCycleTimeInMS*nDimCmdCycleTimeFactor, 
	bRunTuning:= bRunTuning, 
	bOccupiedRoom=> bOccupiedRoom, 
	bError_Prim=> , 
	nError_Prim=> , 
	stTuneData:=stTuneData , 
	stPirSensorData:= stPirSensorData, 
	stLiveData:= stLiveData);
END_ACTION

ACTION A_ModbusComm:
//Manage data for modbus communication

//Manage data for read-only in PLC
stRoomDataPLC.bPirActive			:= stPirSensorData.bPrc;
stRoomDataPLC.uiActLuxLevel			:= TO_UINT(TRUNC(stPirSensorData.fBrightness));
stRoomDataPLC.uiActLightLevelPct	:= TO_UINT(TRUNC(fbLys.fbBallast.fActlLgtLvl_Prim));
		//stRoomDataPLC.uiActLightLevelPct	:= TO_UINT(TRUNC(fbLys.fbBallast.fActlLgtLvl_Prim)); //if only one group light control
stRoomDataPLC.uiBallastOnHours		:= uiBallastOnHours_MB; //The calculation for BallastOnHours is stored directly to the MB register below


//Assign data for read-only to MB registers
bPirActive_MB			:= stRoomDataPLC.bPirActive;
uiActLuxLevel_MB		:= stRoomDataPLC.uiActLuxLevel;
uiActLightLevelPct_MB	:= stRoomDataPLC.uiActLightLevelPct;

	//calculate BallastOnHours
	fbBallastOnHours(
		bEnableHourCount	:= bEnableHourCount,
		bPauseCount			:= fbLys.fbLightCtrl.bOffZone1,
		uiOnHours			:= uiBallastOnHours_MB,			//OnHours is updated here
		byOverflowCount		:= byOnHoursOverflowCount);


//Manage data for read/write for both PLC and MB registers
fbWriteSPLuxLevel(	nMaxValOut	:= uiMaxLuxLevel,
					nValIn1		:= uiSPLuxLevel_MB,		//nValIn1 takes priotity in case of download or restart
					nValIn2		:= stRoomDataPLC.uiSpLuxLevel,
					nValOut		=> uiLuxOn
				);


fbWritePirDelayTIme(	nMaxValOut	:= uiMaxPirOffMinutes,
						nValIn1		:= uiPirOffDelayTime_MB,		//nValIn1 takes priotity in case of download or restart
						nValIn2		:= stRoomDataPLC.uiPirOffDelayTime,
						nValOut		=> uiPirOffMinutes
					);
					

//Convert read/write modbus data to appropriate datatypes in PLC
fLuxOn	:= TO_REAL(uiLuxOn);			
tPIROff	:= TO_TIME(uiPirOffMinutes*udTimeScaling); //Time conversion defaults to ms

fLuxDim	:= TO_REAL(stRoomDataPLC.uiSpDimLuxLevel);			
tPIRDim	:= TO_TIME(stRoomDataPLC.uiPirDimDelayTime*udTimeScaling); //Time conversion defaults to ms
END_ACTION

ACTION A_Sensor:

fbSensor.ipCommunication := P_DALI_Background.arrfbKL6821Communication[Sesnor_DALI_LINE_NUM];

fbSensor(
	byShrtAdr:= bySensorAddr, 
	bInitialize:= bInitialize, 
	DALI_LINE_NUM:= Sesnor_DALI_LINE_NUM, 
 	//bCancelHoldTimerOccupancy:= bCancelHoldTimerOccupancy, 
	stSensorSetup := stDaliSensorSetup,
	bInitErr=> bInitErr, 
	bInitDone=> bInitDone,
	stPirSensorData:= stPirSensorData, 
	arrSensorScales:= arrSensorScales);
END_ACTION

END_PROGRAM

// ---- POUs/Alle_Rum/Rum_Med_DALI_Pir/Rum_1_111D/P_Rum_1_111D.TcPOU
PROGRAM P_Rum_1_111D
VAR
//Light

	fbLys		: FB_Light_Type_A;
	
	stDaliSetup	: SH_Light.ST_DALI_RoomSetup := (		byShrtAdr_Prim := 52, 
														byGrpAdr_Prim := 8, 
														eMod_Prim := E_DALIAddressType.Group, 
														//byShrtAdr_Sec := 1, 
														//byGrpAdr_Sec := 1, 
														//eMod_Sec := E_DALIAddressType.Short, 
														//byShrtAdr_Supl := 1, 
														DALI_LINE_NUM_PRIM := 2, 
														DALI_LINE_NUM_SEC := 0, 
														DALI_LINE_NUM_SUPL := 0);
	stLiveData				: SH_Light.ST_LiveData;
	bRunTuning					: BOOL;
	
	bTopButtonZone1				: BOOL;
	bTopButtonZone1_Visu		: BOOL;
	bBottomButtonZone1			: BOOL;
	bBottomButtonZone1_Visu	    : BOOL;
	bButtonZone2				: BOOL;
	bNeighborRoomsPir		    : BOOL;
	fLuxOn				     	: REAL;
	fLuxDim						: REAL;
	tPIRDim						: TIME;
	tPIROff						: TIME;
	fOffsetSec					: REAL := 20;
	bOccupiedRoom			    : BOOL;



// Sensor Settings	
	fbSensor					: SH_Light.FB_NIKO_P46xx_1Pcs;
	//fbSensor					: SH_Light.FB_NIKO_P46xx_2Pcs;
	bySensorAddr				: BYTE := 13;
	//arrSensorAddr				: ARRAY[1..2] OF BOOL;
	bInitialize					: BOOL := TRUE;
	stDaliSensorSetup			: ST_DALI_NIKOP46SetupData := (
																nSensitivityPIRSegmentA := arrSensitivityOccupancy[1],
																nSensitivityPIRSegmentB := arrSensitivityOccupancy[2],
																nSensitivityPIRSegmentC := arrSensitivityOccupancy[3]);

	bInitErr				: BOOL;
	bInitDone				: BOOL;
	//arrInitErr					: ARRAY [1..2] OF BOOL;
	//arrInitDone					: ARRAY [1..2] OF BOOL;
	arrSensorScales				: ARRAY [1..10] OF SH_Light.ST_DALI_SensorScaleMode := [	(fMeassureMaxSensor := fMeassure_Zone10, fReadMaxSensor := fRead_Zone10),
																						9(())];
	bCancelHoldTimerOccupancy	: BOOL;
(*	eEventPriorityOccupancy		: E_DALIEventPriority := E_DALIEVENTPRIORITY.Middle;
	nHoldTimerOccupancy			: WORD := 5; // Value in s. 	
	nReportTimerOccupancy		: BYTE := 120; // Value in s, Preset manufacturer value
	nDeadtimeTimerOccupancy		: WORD := 100; // Value in ms, Predefined Value of DALI Standard
	bCancelHoldTimerOccupancy	: BOOL;
	nSensitivityOccupancy		: BYTE:= 3; //setting Sensivity (0..4) 0 (Off), 1 (Min), 2(Low), 3(High) and 4 (Max)

	bEnableLuxEvent				: BOOL;
	eEventPriorityBrightness	: E_DALIEventPriority := E_DALIEVENTPRIORITY.Middle;
	nDeadtimeTimerBrightness	: WORD := 1500; // Value in ms, Predefined Value of DALI Standard
	nHysteresisBrightness		: BYTE := 2; // Value in %
	nHysteresisMinBrightness	: BYTE := 10; // Absolute Value, depending on the manufacturer specific resolution
	nReportTimerBrightness		: BYTE := 120; // Value in s, Preset manufacturer value
*)

	//ModbusComm setup
	
	fbWriteSPLuxLevel			: SH_Light.FB_TwoVal_SelectOne_RTrigChange;
	fbWritePirDelayTIme		: SH_Light.FB_TwoVal_SelectOne_RTrigChange;
	stRoomDataPLC				: SH_Light.ST_RoomDataPLC	:=	(
																	uiPirOffDelayTime	:= 30,
																	uiSpLuxLevel		:= 500,
																	uiPirDimDelayTime	:= 15,
																	uiSpDimLuxLevel		:= 200);
																	
	fbBallastOnHours				: SH_Light.FB_CountOnHours;
	bEnableHourCount			: BOOL := TRUE;
	
	//Non-persistent modbus data
	bPirActive_MB					AT %MX500.0	: BOOL;				//bPirLys i gammel kode
	uiActLuxLevel_MB			    AT %MB504	: UINT;				//intHMIAktueltLux i gammel kode
	uiActLightLevelPct_MB	        AT %MB508	: UINT;				//intDALI_Gruppe1_Lysniveau i gammel kode
	
	//For Conversion
	uiPirOffMinutes						: UINT;
	udTimeScaling						: UDINT := 60000;
	uiLuxOn								: UINT;
	
	//max values checks
	uiMaxLuxLevel						: UINT := 1023;
	uiMaxPirOffMinutes				    : UINT := 180;

	
END_VAR

VAR CONSTANT
	Sesnor_DALI_LINE_NUM: BYTE := 2;
	DALI_LINE_NUM_LIGHT: BYTE := 2;
	DALI_LINE_NUM_PENDANTS	            : BYTE := 0; //0=ingen pendler	
	arrSensitivityOccupancy				: ARRAY[1..3] OF BYTE := [4,4,4]; //sensitivitet for sensor

END_VAR
VAR PERSISTENT
	stPirSensorData: SH_Light.ST_DALI_Sensor;
	stTuneData: SH_Light.ST_TuneData_EX;
	
	uiPirOffDelayTime_MB	AT %MB502	: UINT;				//ntHMI_Pir_SetValue i gammel kode
	uiSPLuxLevel_MB			AT %MB506	: UINT;				//intHMI_Lux_SetValue i gammel kode
	uiBallastOnHours_MB		AT %MB510	: UINT;				//dintHMILysbraendtimer1 i gammel kode
	byOnHoursOverflowCount				: BYTE;   

END_VAR

A_Buttons();
A_LightCtrl();
A_Sensor();
A_Modbuscomm();

ACTION A_Buttons:
bTopButtonZone1		:= bTopButtonZone1_Visu;
bBottomButtonZone1	:= bBottomButtonZone1_Visu;
END_ACTION

ACTION A_LightCtrl:

fbLys(
	nZoneID:= 1, 
	bButtonZone1:= bTopButtonZone1,
	bBottomButtonZone1 := bBottomButtonZone1, 
	bButtonZone2:= bButtonZone2, 
	fLuxOn:= fLuxOn, 
	fLuxDim:= fLuxDim, 
	tPIRDim:= tPIRDim, 
	tPIROff:= tPIROff, 
	fOffsetSec:= fOffsetSec, 
	bReInit:= , 
	stDaliSetup:= stDaliSetup, 
	ipCommunication_Prim:= P_DALI_Background.arrfbKL6821Communication[DALI_LINE_NUM_LIGHT], 
	//ipCommunication_Sec:= P_DALI_Background.arrfbKL6821Communication[DALI_LINE_NUM_LIGHT], 
	//ipCommunication_Supl:= P_DALI_Background.arrfbKL6821Communication[DALI_LINE_NUM_LIGHT], 
	fMinOutputPowerLevelRoom:= 15, 
	fMaxOutputPowerLevelRoom:= 100, 
	nCycleTimeInMS:=  SH_Light.DALI_Param.nPlcTaskCycleTimeInMS*nDimCmdCycleTimeFactor , 
	bRunTuning:= bRunTuning, 
	bOccupiedRoom=> bOccupiedRoom, 
	bError_Prim=> , 
	nError_Prim=> , 
	stTuneData:=stTuneData , 
	stPirSensorData:= stPirSensorData, 
	stLiveData:= stLiveData);
END_ACTION

ACTION A_ModbusComm:
//Manage data for modbus communication

//Manage data for read-only in PLC
stRoomDataPLC.bPirActive			:= stPirSensorData.bPrc;
stRoomDataPLC.uiActLuxLevel			:= TO_UINT(TRUNC(stPirSensorData.fBrightness));
stRoomDataPLC.uiActLightLevelPct	:= TO_UINT(TRUNC(fbLys.fbBallast.fActlLgtLvl_Prim));
		//stRoomDataPLC.uiActLightLevelPct	:= TO_UINT(TRUNC(fbLys.fbBallast.fActlLgtLvl_Prim)); //if only one group light control
stRoomDataPLC.uiBallastOnHours		:= uiBallastOnHours_MB; //The calculation for BallastOnHours is stored directly to the MB register below


//Assign data for read-only to MB registers
bPirActive_MB			:= stRoomDataPLC.bPirActive;
uiActLuxLevel_MB		:= stRoomDataPLC.uiActLuxLevel;
uiActLightLevelPct_MB	:= stRoomDataPLC.uiActLightLevelPct;

	//calculate BallastOnHours
	fbBallastOnHours(
		bEnableHourCount	:= bEnableHourCount,
		bPauseCount			:= fbLys.fbLightCtrl.bOffZone1,
		uiOnHours			:= uiBallastOnHours_MB,			//OnHours is updated here
		byOverflowCount		:= byOnHoursOverflowCount);


//Manage data for read/write for both PLC and MB registers
fbWriteSPLuxLevel(	nMaxValOut	:= uiMaxLuxLevel,
					nValIn1		:= uiSPLuxLevel_MB,		//nValIn1 takes priotity in case of download or restart
					nValIn2		:= stRoomDataPLC.uiSpLuxLevel,
					nValOut		=> uiLuxOn
				);


fbWritePirDelayTIme(	nMaxValOut	:= uiMaxPirOffMinutes,
						nValIn1		:= uiPirOffDelayTime_MB,		//nValIn1 takes priotity in case of download or restart
						nValIn2		:= stRoomDataPLC.uiPirOffDelayTime,
						nValOut		=> uiPirOffMinutes
					);
					

//Convert read/write modbus data to appropriate datatypes in PLC
fLuxOn	:= TO_REAL(uiLuxOn);			
tPIROff	:= TO_TIME(uiPirOffMinutes*udTimeScaling); //Time conversion defaults to ms

fLuxDim	:= TO_REAL(stRoomDataPLC.uiSpDimLuxLevel);			
tPIRDim	:= TO_TIME(stRoomDataPLC.uiPirDimDelayTime*udTimeScaling); //Time conversion defaults to ms
END_ACTION

ACTION A_Sensor:

fbSensor.ipCommunication := P_DALI_Background.arrfbKL6821Communication[Sesnor_DALI_LINE_NUM];

fbSensor(
	byShrtAdr:= bySensorAddr, 
	bInitialize:= bInitialize, 
	DALI_LINE_NUM:= Sesnor_DALI_LINE_NUM, 
 	//bCancelHoldTimerOccupancy:= bCancelHoldTimerOccupancy, 
	stSensorSetup := stDaliSensorSetup,
	bInitErr=> bInitErr, 
	bInitDone=> bInitDone,
	stPirSensorData:= stPirSensorData, 
	arrSensorScales:= arrSensorScales);
END_ACTION

END_PROGRAM

// ---- POUs/Alle_Rum/Trapper/P_Trappe_T1.TcPOU
PROGRAM P_Trappe_T1
VAR
	bDigitalPir				AT%I*	: BOOL;
	bTrappelysNC		AT%Q*	: BOOL;
	
	fbTon_Off				: TON;
	tPirTidOff				: TIME;
	tPirTidOff_PLC	: TIME := T#1M;
	bIngenAktivitet		: BOOL;
	bTrappeLys			: BOOL;
	
	//Modbus data Read
	bTrappeAktivitet		: BOOL;
	//Modbus data Read/Wrtite
	bPirTidOff_MB			: TIME;
	
END_VAR


bIngenAktivitet	:= NOT bDigitalPir;
tPirTidOff		:= tPirTidOff_PLC;

fbTon_Off(IN:= bIngenAktivitet, PT:= tPirTidOff);

IF bDigitalPir  THEN
	bTrappeLys := TRUE;
END_IF
IF fbTon_Off.Q THEN
	bTrappeLys := FALSE;
END_IF

bTrappelysNC 	:= NOT bTrappeLys;

END_PROGRAM

// ---- POUs/DALI/DALI_Setup/FBs/FB_Part102MemoryPages.TcPOU
FUNCTION_BLOCK FB_Part102MemoryPages
VAR_INPUT
	ipDALICommunication				:	I_DALICommunication;
END_VAR
VAR_OUTPUT
	bBusy							:	BOOL;
END_VAR
VAR
	{region "Visu"}
	bRead							:	BOOL;
	bWrite							:	BOOL;
	bHideWaitSymbol					:	BOOL := TRUE;
	aMemoryBank						:	ARRAY [0..254] OF ST_DALIMemoryBank;
	{endregion}
	aValues							:	ARRAY [0..254] OF BYTE;
	nStep							:	INT;
	nAddress						:	BYTE;
	nMemoryBank						:	BYTE;
	nOffset							:	INT := 0;
	aNoValue						:	ARRAY [0..254] OF BOOL;
	nNoValue						:	BYTE;

	fb103StartQuiescentMode			:	FB_DALI103StartQuiescentMode(0);
	fb103StopQuiescentMode			:	FB_DALI103StopQuiescentMode(0);
	fb102ReadMemoryLocation			:	FB_DALI102ReadMemoryLocation(0);
	fb102WriteMemoryLocationNoReply	:	FB_DALI102WriteMemoryLocationNoReply(0);
END_VAR

IF (bRead AND (nStep = 0)) THEN
	nStep := 5;
	bRead := FALSE;
	bHideWaitSymbol := FALSE;
END_IF

IF (bWrite AND (nStep = 0)) THEN
	nStep := 1000;
	bWrite := FALSE;
	bHideWaitSymbol := FALSE;
END_IF

{region "Manage Dialog Selection}
IF (nStep = 0) THEN
	bBusy := FALSE;
ELSE
	bBusy := TRUE;
END_IF
{endregion}

{region "Execute Commands"}
CASE nStep OF
0:
{region "Init"}
	bRead := FALSE;
	bWrite := FALSE;
	bHideWaitSymbol := TRUE;

	fb103StartQuiescentMode.ipDALICommunication := ipDALICommunication;
	fb103StopQuiescentMode.ipDALICommunication := ipDALICommunication;
	fb102ReadMemoryLocation.ipDALICommunication := ipDALICommunication;
	fb102WriteMemoryLocationNoReply.ipDALICommunication := ipDALICommunication;
{endregion}
{region "Read"}
5:
{region "Start Qiescent Mode"}
	fb103StartQuiescentMode(bStart := TRUE,
							eAddressType := Tc3_DALI.E_DALIAddressType.Broadcast,
							eCommandPriority := Tc3_DALI.E_DALICommandPriority.Middle);
	IF (NOT fb103StartQuiescentMode.bBusy) THEN
		fb103StartQuiescentMode(bStart:= FALSE);
		nStep := 10;
	END_IF
{endregion}
10:
{region "Read values from selected memory bank"}
	fb102ReadMemoryLocation(bStart := TRUE,
							nAddress := nAddress,
							eAddressType := Tc3_DALI.E_DALIAddressType.Short,
							eCommandPriority := Tc3_DALI.E_DALICommandPriority.Middle,
							nMemoryBank := nMemoryBank,
							nOffset := INT_TO_BYTE(nOffset),
							nValue => aValues[nOffset]);
	IF (NOT fb102ReadMemoryLocation.bBusy) THEN
		aMemoryBank[nOffset].nValueDec := aValues[nOffset];
		aMemoryBank[nOffset].nValueHex := CONCAT('0x', BYTE_TO_HEXSTR(aValues[nOffset], 2, FALSE));
		nOffset	:= nOffset + 1;
		IF (nOffset > aValues[0]) THEN
			nOffset := 0;
			nStep := 20;
		END_IF
		fb102ReadMemoryLocation(bStart := FALSE);
	END_IF
{endregion}
20:
{region "Hide unused rows in table"}
	FOR nNoValue := (aValues[0] + 1) TO 254 DO
		aNoValue[nNoValue] := TRUE;
	END_FOR
	FOR nNoValue := 0 TO (aValues[0]) DO
		aNoValue[nNoValue] := FALSE;
	END_FOR
nStep := 25;
{endregion}
25:
{region "Stop Qiescent Mode"}
	fb103StopQuiescentMode(	bStart := TRUE,
							eAddressType := Tc3_DALI.E_DALIAddressType.Broadcast,
							eCommandPriority := Tc3_DALI.E_DALICommandPriority.Middle);
	IF (NOT fb103StopQuiescentMode.bBusy) THEN
		fb103StopQuiescentMode(bStart:= FALSE);
		nStep := 0;
	END_IF
{endregion}	
1000:
{region "Change Value"}
	IF (nMemoryBank >= 1) THEN
		aValues[nOffset] := aMemoryBank[nOffset].nValueDec;
		fb102WriteMemoryLocationNoReply(bStart := TRUE,
										nAddress := nAddress,
										eAddressType := Tc3_DALI.E_DALIAddressType.Short,
										eCommandPriority := Tc3_DALI.E_DALICommandPriority.Middle,
										nMemoryBank := nMemoryBank,
										nOffset := INT_TO_BYTE(nOffset),
										nValue := aValues[nOffset]);
		IF (NOT fb102WriteMemoryLocationNoReply.bBusy) THEN
			nStep := 1010;
			fb102WriteMemoryLocationNoReply(bStart := FALSE);
		END_IF
	ELSE 
		nStep := 0;
	END_IF
{endregion}
1010:
{region "read changed value"}
	fb102ReadMemoryLocation(bStart := TRUE,
							nAddress := nAddress,
							eAddressType := Tc3_DALI.E_DALIAddressType.Short,
							eCommandPriority := Tc3_DALI.E_DALICommandPriority.Middle,
							nMemoryBank := nMemoryBank,
							nOffset := INT_TO_BYTE(nOffset),
							nValue => aValues[nOffset]);
	IF (NOT fb102ReadMemoryLocation.bBusy) THEN
		aMemoryBank[nOffset].nValueDec := aValues[nOffset];
		aMemoryBank[nOffset].nValueHex := CONCAT ('0x', BYTE_TO_HEXSTR(aValues[nOffset], 2, FALSE));
		nStep := 0;
		fb102ReadMemoryLocation(bStart := FALSE);
	END_IF
{endregion}
END_CASE

// Filling the according filds of the Array Memory Bank for the HMI display
// Writing clear text for offset description
aMemoryBank[0].sOffset := '0 (0x00)';
aMemoryBank[1].sOffset := '1 (0x01)';
aMemoryBank[2].sOffset := '2 (0x02)';
aMemoryBank[3].sOffset := '3 (0x03)';
aMemoryBank[4].sOffset := '4 (0x04)';
aMemoryBank[5].sOffset := '5 (0x05)';
aMemoryBank[6].sOffset := '6 (0x06)';
aMemoryBank[7].sOffset := '7 (0x07)';
aMemoryBank[8].sOffset := '8 (0x08)';
aMemoryBank[9].sOffset := '9 (0x09)';
aMemoryBank[10].sOffset := '10 (0x0A)';
aMemoryBank[11].sOffset := '11 (0x0B)';
aMemoryBank[12].sOffset := '12 (0x0C)';
aMemoryBank[13].sOffset := '13 (0x0D)';
aMemoryBank[14].sOffset := '14 (0x0E)';
aMemoryBank[15].sOffset := '15 (0x0F)';
aMemoryBank[16].sOffset := '16 (0x10)';
aMemoryBank[17].sOffset := '17 (0x11)';
aMemoryBank[18].sOffset := '18 (0x12)';
aMemoryBank[19].sOffset := '19 (0x13)';
aMemoryBank[20].sOffset := '20 (0x14)';
aMemoryBank[21].sOffset := '21 (0x15)';
aMemoryBank[22].sOffset := '22 (0x16)';
aMemoryBank[23].sOffset := '23 (0x17)';
aMemoryBank[24].sOffset := '24 (0x18)';
aMemoryBank[25].sOffset := '25 (0x19)';
aMemoryBank[26].sOffset := '26 (0x1A)';
aMemoryBank[27].sOffset := '27 (0x1B)';
aMemoryBank[28].sOffset := '28 (0x1C)';
aMemoryBank[29].sOffset := '29 (0x1D)';
aMemoryBank[30].sOffset := '30 (0x1E)';
aMemoryBank[31].sOffset := '31 (0x1F)';
aMemoryBank[32].sOffset := '32 (0x20)';
aMemoryBank[33].sOffset := '33 (0x21)';
aMemoryBank[34].sOffset := '34 (0x22)';
aMemoryBank[35].sOffset := '35 (0x23)';
aMemoryBank[36].sOffset := '36 (0x24)';
aMemoryBank[37].sOffset := '37 (0x25)';
aMemoryBank[38].sOffset := '38 (0x26)';
aMemoryBank[39].sOffset := '39 (0x27)';
aMemoryBank[40].sOffset := '40 (0x28)';
aMemoryBank[41].sOffset := '41 (0x29)';
aMemoryBank[42].sOffset := '42 (0x2A)';
aMemoryBank[42].sOffset := '43 (0x2B)';
aMemoryBank[44].sOffset := '44 (0x2C)';
aMemoryBank[45].sOffset := '45 (0x2D)';
aMemoryBank[46].sOffset := '46 (0x2E)';
aMemoryBank[47].sOffset := '47 (0x2F)';
aMemoryBank[48].sOffset := '48 (0x30)';
aMemoryBank[49].sOffset := '49 (0x31)';
aMemoryBank[50].sOffset := '50 (0x32)';
aMemoryBank[51].sOffset := '51 (0x33)';
aMemoryBank[52].sOffset := '52 (0x34)';
aMemoryBank[53].sOffset := '53 (0x35)';
aMemoryBank[54].sOffset := '54 (0x36)';
aMemoryBank[55].sOffset := '55 (0x37)';
aMemoryBank[56].sOffset := '56 (0x38)';
aMemoryBank[57].sOffset := '57 (0x39)';
aMemoryBank[58].sOffset := '58 (0x3A)';
aMemoryBank[59].sOffset := '59 (0x3B)';
aMemoryBank[60].sOffset := '60 (0x3C)';
aMemoryBank[61].sOffset := '61 (0x3D)';
aMemoryBank[62].sOffset := '62 (0x3F)';
aMemoryBank[63].sOffset := '63 (0x3D)';
aMemoryBank[64].sOffset := '64 (0x40)';
aMemoryBank[65].sOffset := '65 (0x41)';
aMemoryBank[66].sOffset := '66 (0x42)';
aMemoryBank[67].sOffset := '67 (0x43)';
aMemoryBank[68].sOffset := '68 (0x44)';
aMemoryBank[69].sOffset := '69 (0x45)';
aMemoryBank[70].sOffset := '70 (0x46)';
aMemoryBank[71].sOffset := '71 (0x47)';
aMemoryBank[72].sOffset := '72 (0x48)';
aMemoryBank[73].sOffset := '73 (0x49)';
aMemoryBank[74].sOffset := '74 (0x4A)';
aMemoryBank[75].sOffset := '75 (0x4B)';
aMemoryBank[76].sOffset := '76 (0x4C)';
aMemoryBank[77].sOffset := '77 (0x4D)';
aMemoryBank[78].sOffset := '78 (0x4E)';
aMemoryBank[79].sOffset := '79 (0x4F)';
aMemoryBank[80].sOffset := '80 (0x50)';
aMemoryBank[81].sOffset := '81 (0x51)';
aMemoryBank[82].sOffset := '82 (0x52)';
aMemoryBank[83].sOffset := '83 (0x53)';
aMemoryBank[84].sOffset := '84 (0x54)';
aMemoryBank[85].sOffset := '85 (0x55)';
aMemoryBank[86].sOffset := '86 (0x56)';
aMemoryBank[87].sOffset := '87 (0x57)';
aMemoryBank[88].sOffset := '88 (0x58)';
aMemoryBank[89].sOffset := '89 (0x59)';
aMemoryBank[90].sOffset := '90 (0x5A)';
aMemoryBank[91].sOffset := '91 (0x5B)';
aMemoryBank[92].sOffset := '92 (0x5C)';
aMemoryBank[93].sOffset := '93 (0x5D)';
aMemoryBank[94].sOffset := '94 (0x5E)';
aMemoryBank[95].sOffset := '95 (0x5F)';
aMemoryBank[96].sOffset := '96 (0x60)';
aMemoryBank[97].sOffset := '97 (0x61)';
aMemoryBank[98].sOffset := '98 (0x62)';
aMemoryBank[99].sOffset := '99 (0x63)';
aMemoryBank[100].sOffset := '100 (0x64)';
aMemoryBank[101].sOffset := '101 (0x65)';
aMemoryBank[102].sOffset := '102 (0x66)';
aMemoryBank[103].sOffset := '103 (0x67)';
aMemoryBank[104].sOffset := '104 (0x68)';
aMemoryBank[105].sOffset := '105 (0x69)';
aMemoryBank[106].sOffset := '106 (0x6A)';
aMemoryBank[107].sOffset := '107 (0x6B)';
aMemoryBank[108].sOffset := '108 (0x6C)';
aMemoryBank[109].sOffset := '109 (0x6D)';
aMemoryBank[110].sOffset := '110 (0x6E)';
aMemoryBank[111].sOffset := '111 (0x6F)';
aMemoryBank[112].sOffset := '112 (0x70)';
aMemoryBank[113].sOffset := '113 (0x71)';
aMemoryBank[114].sOffset := '114 (0x72)';
aMemoryBank[115].sOffset := '115 (0x73)';
aMemoryBank[116].sOffset := '116 (0x74)';
aMemoryBank[117].sOffset := '117 (0x75)';
aMemoryBank[118].sOffset := '118 (0x76)';
aMemoryBank[119].sOffset := '119 (0x77)';
aMemoryBank[120].sOffset := '120 (0x78)';
aMemoryBank[121].sOffset := '121 (0x79)';
aMemoryBank[122].sOffset := '122 (0x7A)';
aMemoryBank[123].sOffset := '123 (0x7B)';
aMemoryBank[124].sOffset := '124 (0x7C)';
aMemoryBank[125].sOffset := '125 (0x7D)';
aMemoryBank[126].sOffset := '126 (0x7E)';
aMemoryBank[127].sOffset := '127 (0x7F)';
aMemoryBank[128].sOffset := '128 (0x80)';
aMemoryBank[129].sOffset := '129 (0x81)';
aMemoryBank[130].sOffset := '130 (0x82)';
aMemoryBank[131].sOffset := '131 (0x83)';
aMemoryBank[132].sOffset := '132 (0x84)';
aMemoryBank[133].sOffset := '133 (0x85)';
aMemoryBank[134].sOffset := '134 (0x86)';
aMemoryBank[135].sOffset := '135 (0x87)';
aMemoryBank[136].sOffset := '136 (0x88)';
aMemoryBank[137].sOffset := '137 (0x89)';
aMemoryBank[138].sOffset := '138 (0x8A)';
aMemoryBank[139].sOffset := '139 (0x8B)';
aMemoryBank[140].sOffset := '140 (0x8C)';
aMemoryBank[141].sOffset := '141 (0x8D)';
aMemoryBank[142].sOffset := '142 (0x8E)';
aMemoryBank[143].sOffset := '143 (0x8F)';
aMemoryBank[144].sOffset := '144 (0x90)';
aMemoryBank[145].sOffset := '145 (0x91)';
aMemoryBank[146].sOffset := '146 (0x92)';
aMemoryBank[147].sOffset := '147 (0x93)';
aMemoryBank[148].sOffset := '148 (0x94)';
aMemoryBank[149].sOffset := '149 (0x95)';
aMemoryBank[150].sOffset := '150 (0x96)';
aMemoryBank[151].sOffset := '151 (0x97)';
aMemoryBank[152].sOffset := '152 (0x98)';
aMemoryBank[153].sOffset := '153 (0x99)';
aMemoryBank[154].sOffset := '154 (0x9A)';
aMemoryBank[155].sOffset := '155 (0x9B)';
aMemoryBank[156].sOffset := '156 (0x9C)';
aMemoryBank[157].sOffset := '157 (0x9D)';
aMemoryBank[158].sOffset := '158 (0x9E)';
aMemoryBank[159].sOffset := '159 (0x9F)';
aMemoryBank[160].sOffset := '160 (0xA0)';
aMemoryBank[161].sOffset := '161 (0xA1)';
aMemoryBank[162].sOffset := '162 (0xA2)';
aMemoryBank[163].sOffset := '163 (0xA3)';
aMemoryBank[164].sOffset := '164 (0xA4)';
aMemoryBank[165].sOffset := '165 (0xA5)';
aMemoryBank[166].sOffset := '166 (0xA6)';
aMemoryBank[167].sOffset := '167 (0xA7)';
aMemoryBank[168].sOffset := '168 (0xA8)';
aMemoryBank[169].sOffset := '169 (0xA9)';
aMemoryBank[170].sOffset := '170 (0xAA)';
aMemoryBank[171].sOffset := '171 (0xAB)';
aMemoryBank[172].sOffset := '172 (0xAC)';
aMemoryBank[173].sOffset := '173 (0xAD)';
aMemoryBank[174].sOffset := '174 (0xAE)';
aMemoryBank[175].sOffset := '175 (0xAF)';
aMemoryBank[176].sOffset := '176 (0xB0)';
aMemoryBank[177].sOffset := '177 (0xB1)';
aMemoryBank[178].sOffset := '178 (0xB2)';
aMemoryBank[179].sOffset := '179 (0xB3)';
aMemoryBank[180].sOffset := '180 (0xB4)';
aMemoryBank[181].sOffset := '181 (0xB5)';
aMemoryBank[182].sOffset := '182 (0xB6)';
aMemoryBank[183].sOffset := '183 (0xB7)';
aMemoryBank[184].sOffset := '184 (0xB8)';
aMemoryBank[185].sOffset := '185 (0xB9)';
aMemoryBank[186].sOffset := '186 (0xBA)';
aMemoryBank[187].sOffset := '187 (0xBB)';
aMemoryBank[188].sOffset := '188 (0xBC)';
aMemoryBank[189].sOffset := '189 (0xBD)';
aMemoryBank[190].sOffset := '190 (0xDE)';
aMemoryBank[191].sOffset := '191 (0xBF)';
aMemoryBank[192].sOffset := '192 (0xC0)';
aMemoryBank[193].sOffset := '193 (0xC1)';
aMemoryBank[194].sOffset := '194 (0xC3)';
aMemoryBank[195].sOffset := '195 (0xC4)';
aMemoryBank[196].sOffset := '196 (0xC5)';
aMemoryBank[197].sOffset := '197 (0xC6)';
aMemoryBank[198].sOffset := '198 (0xC7)';
aMemoryBank[199].sOffset := '199 (0xC8)';
aMemoryBank[200].sOffset := '200 (0xC9)';
aMemoryBank[201].sOffset := '201 (0xCA)';
aMemoryBank[202].sOffset := '202 (0xCB)';
aMemoryBank[203].sOffset := '203 (0xCC)';
aMemoryBank[204].sOffset := '204 (0xCD)';
aMemoryBank[205].sOffset := '205 (0xCE)';
aMemoryBank[206].sOffset := '206 (0xCF)';
aMemoryBank[207].sOffset := '207 (0xD0)';
aMemoryBank[208].sOffset := '208 (0xD1)';
aMemoryBank[209].sOffset := '209 (0xD2)';
aMemoryBank[210].sOffset := '210 (0xD3)';
aMemoryBank[211].sOffset := '211 (0xD4)';
aMemoryBank[212].sOffset := '212 (0xD5)';
aMemoryBank[213].sOffset := '213 (0xD6)';
aMemoryBank[214].sOffset := '214 (0xD7)';
aMemoryBank[215].sOffset := '215 (0xD8)';
aMemoryBank[216].sOffset := '216 (0xD9)';
aMemoryBank[217].sOffset := '217 (0xDA)';
aMemoryBank[218].sOffset := '218 (0xDB)';
aMemoryBank[219].sOffset := '219 (0xDC)';
aMemoryBank[220].sOffset := '220 (0xDD)';
aMemoryBank[221].sOffset := '221 (0xDE)';
aMemoryBank[222].sOffset := '222 (0xDF)';
aMemoryBank[223].sOffset := '223 (0xE0)';
aMemoryBank[224].sOffset := '224 (0xE1)';
aMemoryBank[225].sOffset := '225 (0xE2)';
aMemoryBank[226].sOffset := '226 (0xE3)';
aMemoryBank[227].sOffset := '227 (0xE4)';
aMemoryBank[228].sOffset := '228 (0xE5)';
aMemoryBank[229].sOffset := '229 (0xE6)';
aMemoryBank[230].sOffset := '230 (0xE7)';
aMemoryBank[231].sOffset := '231 (0xE8)';
aMemoryBank[232].sOffset := '232 (0xE9)';
aMemoryBank[233].sOffset := '233 (0xEA)';
aMemoryBank[234].sOffset := '234 (0xEB)';
aMemoryBank[235].sOffset := '235 (0xEC)';
aMemoryBank[236].sOffset := '236 (0xED)';
aMemoryBank[237].sOffset := '237 (0xEE)';
aMemoryBank[238].sOffset := '238 (0xEF)';
aMemoryBank[239].sOffset := '239 (0xF0)';
aMemoryBank[240].sOffset := '240 (0xF1)';
aMemoryBank[241].sOffset := '241 (0xF2)';
aMemoryBank[242].sOffset := '242 (0xF3)';
aMemoryBank[243].sOffset := '243 (0xF4)';
aMemoryBank[244].sOffset := '244 (0xF5)';
aMemoryBank[245].sOffset := '245 (0xF6)';
aMemoryBank[246].sOffset := '246 (0xF7)';
aMemoryBank[247].sOffset := '247 (0xF8)';
aMemoryBank[248].sOffset := '248 (0xF9)';
aMemoryBank[249].sOffset := '249 (0xFA)';
aMemoryBank[250].sOffset := '250 (0xFB)';
aMemoryBank[251].sOffset := '251 (0xFC)';
aMemoryBank[252].sOffset := '252 (0xFD)';
aMemoryBank[253].sOffset := '253 (0xFE)';
aMemoryBank[254].sOffset := '254 (0xFF)';

